	// ===== bw200-C2 =====
	REGION J2.1.2
	    //J2.1.2
	    DB_UDI.EmptyLine.Fault.Stop.Conveyor[_."J2.1.2"] :=
	    _."ASiGW-MCC001-bw200-C2: Input"."Error J2.1.2" OR
	    _."ASiGW-MCC001-bw200-C2: ConfigErr".Slave."16A" OR
	    _."ASiGW-MCC001-bw200-C2: PeriErr".Slave."16A" OR
	    _.Global.IDB_HardwareDiag."BW-ASi -10.106.129.200".CommunicationError;
	    
	END_REGION
	
	// ===== bw200-C2 =====
	REGION J2.1.3
	    //J2.1.3
	    DB_UDI.EmptyLine.Fault.Stop.Conveyor[_."J2.1.3"] :=
	    _."ASiGW-MCC001-bw200-C2: Input"."Error J2.1.3" OR
	    _."ASiGW-MCC001-bw200-C2: ConfigErr".Slave."17A" OR
	    _."ASiGW-MCC001-bw200-C2: PeriErr".Slave."17A" OR
	    _.Global.IDB_HardwareDiag."BW-ASi -10.106.129.200".CommunicationError;
	    
	END_REGION
	
	// ===== bw200-C2 =====
	REGION J2.1.4
	    //J2.1.4
	    DB_UDI.EmptyLine.Fault.Stop.Conveyor[_."J2.1.4"] :=
	    _."ASiGW-MCC001-bw200-C2: Input"."Error J2.1.4" OR
	    _."ASiGW-MCC001-bw200-C2: ConfigErr".Slave."17A" OR
	    _."ASiGW-MCC001-bw200-C2: PeriErr".Slave."17A" OR
	    _.Global.IDB_HardwareDiag."BW-ASi -10.106.129.200".CommunicationError;
	    
	END_REGION
	
	// ===== bw200-C2 =====
	REGION J2.1.5
	    //J2.1.5
	    DB_UDI.EmptyLine.Fault.Stop.Conveyor[_."J2.1.5"] :=
	    _."ASiGW-MCC001-bw200-C2: Input"."Error J2.1.5" OR
	    _."ASiGW-MCC001-bw200-C2: ConfigErr".Slave."18A" OR
	    _."ASiGW-MCC001-bw200-C2: PeriErr".Slave."18A" OR
	    _.Global.IDB_HardwareDiag."BW-ASi -10.106.129.200".CommunicationError;
	    
	END_REGION
	
	// ===== bw200-C2 =====
	REGION J2.1.6
	    //J2.1.6
	    DB_UDI.EmptyLine.Fault.Stop.Conveyor[_."J2.1.6"] :=
	    _."ASiGW-MCC001-bw200-C2: Input"."Error J2.1.6" OR
	    _."ASiGW-MCC001-bw200-C2: ConfigErr".Slave."18A" OR
	    _."ASiGW-MCC001-bw200-C2: PeriErr".Slave."18A" OR
	    _.Global.IDB_HardwareDiag."BW-ASi -10.106.129.200".CommunicationError;
	    
	END_REGION
	
	// ===== bw200-C2 =====
	REGION J2.1.7
	    //J2.1.7
	    DB_UDI.EmptyLine.Fault.Stop.Conveyor[_."J2.1.7"] :=
	    _."ASiGW-MCC001-bw200-C2: Input"."Error J2.1.7" OR
	    _."ASiGW-MCC001-bw200-C2: ConfigErr".Slave."19A" OR
	    _."ASiGW-MCC001-bw200-C2: PeriErr".Slave."19A" OR
	    _.Global.IDB_HardwareDiag."BW-ASi -10.106.129.200".CommunicationError;
	    
	END_REGION
	
	// ===== bw200-C2 =====
	REGION J2.1.8
	    //J2.1.8
	    DB_UDI.EmptyLine.Fault.Stop.Conveyor[_."J2.1.8"] :=
	    _."ASiGW-MCC001-bw200-C2: Input"."Error J2.1.8" OR
	    _."ASiGW-MCC001-bw200-C2: ConfigErr".Slave."19A" OR
	    _."ASiGW-MCC001-bw200-C2: PeriErr".Slave."19A" OR
	    _.Global.IDB_HardwareDiag."BW-ASi -10.106.129.200".CommunicationError;
	    
	END_REGION
	
	// ===== bw200-C2 =====
	REGION J2.1.9
	    //J2.1.9
	    DB_UDI.EmptyLine.Fault.Stop.Conveyor[_."J2.1.9"] :=
	    _."ASiGW-MCC001-bw200-C2: Input"."Error J2.1.9" OR
	    _."ASiGW-MCC001-bw200-C2: ConfigErr".Slave."20A" OR
	    _."ASiGW-MCC001-bw200-C2: PeriErr".Slave."20A" OR
	    _.Global.IDB_HardwareDiag."BW-ASi -10.106.129.200".CommunicationError;
	    
	END_REGION
	
	// ===== bw200-C2 =====
	REGION J2.1.10
	    //J2.1.10
	    DB_UDI.EmptyLine.Fault.Stop.Conveyor[_."J2.1.10"] :=
	    _."ASiGW-MCC001-bw200-C2: Input"."Error J2.1.10" OR
	    _."ASiGW-MCC001-bw200-C2: ConfigErr".Slave."20A" OR
	    _."ASiGW-MCC001-bw200-C2: PeriErr".Slave."20A" OR
	    _.Global.IDB_HardwareDiag."BW-ASi -10.106.129.200".CommunicationError;
	    
	END_REGION
	
	// ===== bw200-C2 =====
	REGION J2.1.11
	    //J2.1.11
	    DB_UDI.EmptyLine.Fault.Stop.Conveyor[_."J2.1.11"] :=
	    _."ASiGW-MCC001-bw200-C2: Input"."Error J2.1.11" OR
	    _."ASiGW-MCC001-bw200-C2: ConfigErr".Slave."21A" OR
	    _."ASiGW-MCC001-bw200-C2: PeriErr".Slave."21A" OR
	    _.Global.IDB_HardwareDiag."BW-ASi -10.106.129.200".CommunicationError;
	    
	END_REGION
	
	// ===== bw200-C2 =====
	REGION J2.1.12
	    //J2.1.12
	    DB_UDI.EmptyLine.Fault.Stop.Conveyor[_."J2.1.12"] :=
	    _."ASiGW-MCC001-bw200-C2: Input"."Error J2.1.12" OR
	    _."ASiGW-MCC001-bw200-C2: ConfigErr".Slave."21A" OR
	    _."ASiGW-MCC001-bw200-C2: PeriErr".Slave."21A" OR
	    _.Global.IDB_HardwareDiag."BW-ASi -10.106.129.200".CommunicationError;
	    
	END_REGION
	
	// ===== bw200-C2 =====
	REGION J2.1.13
	    //J2.1.13
	    DB_UDI.EmptyLine.Fault.Stop.Conveyor[_."J2.1.13"] :=
	    _."ASiGW-MCC001-bw200-C2: Input"."Error J2.1.13" OR
	    _."ASiGW-MCC001-bw200-C2: ConfigErr".Slave."22A" OR
	    _."ASiGW-MCC001-bw200-C2: PeriErr".Slave."22A" OR
	    _.Global.IDB_HardwareDiag."BW-ASi -10.106.129.200".CommunicationError;
	    
	END_REGION
	
	// ===== bw200-C2 =====
	REGION J2.1.14
	    //J2.1.14
	    DB_UDI.EmptyLine.Fault.Stop.Conveyor[_."J2.1.14"] :=
	    _."ASiGW-MCC001-bw200-C2: Input"."Error J2.1.14" OR
	    _."ASiGW-MCC001-bw200-C2: ConfigErr".Slave."22A" OR
	    _."ASiGW-MCC001-bw200-C2: PeriErr".Slave."22A" OR
	    _.Global.IDB_HardwareDiag."BW-ASi -10.106.129.200".CommunicationError;
	    
	END_REGION
	
	// ===== bw200-C2 =====
	REGION J2.1.15
	    //J2.1.15
	    DB_UDI.EmptyLine.Fault.Stop.Conveyor[_."J2.1.15"] :=
	    _."ASiGW-MCC001-bw200-C2: Input"."Error J2.1.15" OR
	    _."ASiGW-MCC001-bw200-C2: ConfigErr".Slave."23A" OR
	    _."ASiGW-MCC001-bw200-C2: PeriErr".Slave."23A" OR
	    _.Global.IDB_HardwareDiag."BW-ASi -10.106.129.200".CommunicationError;
	    
	END_REGION
	
	
	// ===== bw200-C2 =====
	REGION J2.2.1
	    //J2.2.1
	    DB_UDI.EmptyLine.Fault.Stop.Conveyor[_."J2.2.1"] :=
	    _."ASiGW-MCC001-bw200-C2: Input"."Error J2.2.1" OR
	    _."ASiGW-MCC001-bw200-C2: ConfigErr".Slave."23A" OR
	    _."ASiGW-MCC001-bw200-C2: PeriErr".Slave."23A" OR
	    _.Global.IDB_HardwareDiag."BW-ASi -10.106.129.200".CommunicationError;
	    
	END_REGION
	
	// ===== bw200-C2 =====
	REGION J2.2.2
	    //J2.2.2
	    DB_UDI.EmptyLine.Fault.Stop.Conveyor[_."J2.2.2"] :=
	    _."ASiGW-MCC001-bw200-C2: Input"."Error J2.2.2" OR
	    _."ASiGW-MCC001-bw200-C2: ConfigErr".Slave."24A" OR
	    _."ASiGW-MCC001-bw200-C2: PeriErr".Slave."24A" OR
	    _.Global.IDB_HardwareDiag."BW-ASi -10.106.129.200".CommunicationError;
	    
	END_REGION
	
	// ===== bw200-C2 =====
	REGION J2.3.1
	    //J2.3.1
	    DB_UDI.EmptyLine.Fault.Stop.Conveyor[_."J2.3.1"] :=
	    _."ASiGW-MCC001-bw200-C2: ConfigErr".Slave."25A" OR
	    _."ASiGW-MCC001-bw200-C2: PeriErr".Slave."25A" OR
	    _.Global.IDB_HardwareDiag."BW-ASi -10.106.129.200".CommunicationError;
	    
	END_REGION
	
	// ===== bw200-C2 =====
	REGION J2.4.1
	    //J2.4.1 Arm for Merger1
	    DB_UDI.EmptyLine.Fault.Stop.Conveyor[_."J2.4.1"] :=
	    _."ASiGW-MCC001-bw200-C2: Input"."Error J2.4.1" OR
	    _."ASiGW-MCC001-bw200-C2: ConfigErr".Slave."26A" OR
	    _."ASiGW-MCC001-bw200-C2: PeriErr".Slave."26A" OR
	    _.Global.IDB_HardwareDiag."BW-ASi -10.106.129.200".CommunicationError;
	    
	END_REGION
	
	
	// ===== bw143-C1 =====
	REGION J1.2.4 Merger1
	    //J1.2.4 Merger 1
	    DB_UDI.EmptyLine.Fault.Stop.Conveyor[_."J1.2.4"] :=
	    _."ASiGW-MCC001-bw143-C1: Input"."Error J1.2.4" OR
	    _."ASiGW-MCC001-bw143-C1: ConfigErr".Slave."27B" OR
	    _."ASiGW-MCC001-bw143-C1: PeriErr".Slave."27B" OR
	    _.Global.IDB_HardwareDiag."BW-ASi -10.106.129.143".CommunicationError;
	    
	END_REGION
	
	// ===== bw143-C1 =====
	REGION J1.2.5
	    //J1.2.5
	    DB_UDI.EmptyLine.Fault.Stop.Conveyor[_."J1.2.5"] :=
	    _."ASiGW-MCC001-bw143-C1: Input"."Error J1.2.5" OR
	    _."ASiGW-MCC001-bw143-C1: ConfigErr".Slave."27B" OR
	    _."ASiGW-MCC001-bw143-C1: PeriErr".Slave."27B" OR
	    _.Global.IDB_HardwareDiag."BW-ASi -10.106.129.143".CommunicationError;
	    
	END_REGION
	
	
	
	
	
	
	
	
	
	// ===== bw143-C1 =====
	REGION J1.3.1
	    //J1.3.1
	    DB_UDI.EmptyLine.Fault.Stop.Conveyor[_."J1.3.1"] :=
	    _."ASiGW-MCC001-bw143-C1: Input"."Error J1.3.1" OR
	    _."ASiGW-MCC001-bw143-C1: ConfigErr".Slave."17B" OR
	    _."ASiGW-MCC001-bw143-C1: PeriErr".Slave."17B" OR
	    _.Global.IDB_HardwareDiag."BW-ASi -10.106.129.143".CommunicationError;
	    
	END_REGION
	
	// ===== bw143-C1 =====
	REGION J1.3.2
	    //J1.3.2
	    DB_UDI.EmptyLine.Fault.Stop.Conveyor[_."J1.3.2"] :=
	    _."ASiGW-MCC001-bw143-C1: Input"."Error J1.3.2" OR
	    _."ASiGW-MCC001-bw143-C1: ConfigErr".Slave."17B" OR
	    _."ASiGW-MCC001-bw143-C1: PeriErr".Slave."17B" OR
	    _.Global.IDB_HardwareDiag."BW-ASi -10.106.129.143".CommunicationError;
	    
	END_REGION
	
	// ===== bw143-C1 =====
	REGION J1.4.1
	    //J1.4.1
	    DB_UDI.EmptyLine.Fault.Stop.Conveyor[_."J1.4.1"] :=
	    _."ASiGW-MCC001-bw143-C1: Input"."Error J1.4.1" OR
	    _."ASiGW-MCC001-bw143-C1: ConfigErr".Slave."13B" OR
	    _."ASiGW-MCC001-bw143-C1: PeriErr".Slave."13B" OR
	    _.Global.IDB_HardwareDiag."BW-ASi -10.106.129.143".CommunicationError;
	    
	END_REGION
	
	// ===== bw143-C1 =====
	REGION J1.4.2
	    //J1.4.2
	    DB_UDI.EmptyLine.Fault.Stop.Conveyor[_."J1.4.2"] :=
	    _."ASiGW-MCC001-bw143-C1: Input"."Error J1.4.2" OR
	    _."ASiGW-MCC001-bw143-C1: ConfigErr".Slave."13B" OR
	    _."ASiGW-MCC001-bw143-C1: PeriErr".Slave."13B" OR
	    _.Global.IDB_HardwareDiag."BW-ASi -10.106.129.143".CommunicationError;
	    
	END_REGION
	
	// ===== bw143-C1 =====
	REGION J1.4.3
	    //J1.4.3
	    DB_UDI.EmptyLine.Fault.Stop.Conveyor[_."J1.4.3"] :=
	    _."ASiGW-MCC001-bw143-C1: Input"."Error J1.4.3" OR
	    _."ASiGW-MCC001-bw143-C1: ConfigErr".Slave."14B" OR
	    _."ASiGW-MCC001-bw143-C1: PeriErr".Slave."14B" OR
	    _.Global.IDB_HardwareDiag."BW-ASi -10.106.129.143".CommunicationError;
	    
	END_REGION
	
	// ===== bw143-C1 =====
	REGION J1.4.4
	    //J1.4.4
	    DB_UDI.EmptyLine.Fault.Stop.Conveyor[_."J1.4.4"] :=
	    _."ASiGW-MCC001-bw143-C1: Input"."Error J1.4.4" OR
	    _."ASiGW-MCC001-bw143-C1: ConfigErr".Slave."14B" OR
	    _."ASiGW-MCC001-bw143-C1: PeriErr".Slave."14B" OR
	    _.Global.IDB_HardwareDiag."BW-ASi -10.106.129.143".CommunicationError;
	    
	END_REGION
	
	// ===== bw143-C1 =====
	REGION J1.4.5
	    //J1.4.5
	    DB_UDI.EmptyLine.Fault.Stop.Conveyor[_."J1.4.5"] :=
	    _."ASiGW-MCC001-bw143-C1: Input"."Error J1.4.5" OR
	    _."ASiGW-MCC001-bw143-C1: ConfigErr".Slave."15B" OR
	    _."ASiGW-MCC001-bw143-C1: PeriErr".Slave."15B" OR
	    _.Global.IDB_HardwareDiag."BW-ASi -10.106.129.143".CommunicationError;
	    
	END_REGION
	
	// ===== bw143-C1 =====
	REGION J1.4.6
	    //J1.4.6
	    DB_UDI.EmptyLine.Fault.Stop.Conveyor[_."J1.4.6"] :=
	    _."ASiGW-MCC001-bw143-C1: Input"."Error J1.4.6" OR
	    _."ASiGW-MCC001-bw143-C1: ConfigErr".Slave."15B" OR
	    _."ASiGW-MCC001-bw143-C1: PeriErr".Slave."15B" OR
	    _.Global.IDB_HardwareDiag."BW-ASi -10.106.129.143".CommunicationError;
	    
	END_REGION
	
	// ===== bw143-C1 =====
	REGION J1.4.7
	    //J1.4.7
	    DB_UDI.EmptyLine.Fault.Stop.Conveyor[_."J1.4.7"] :=
	    _."ASiGW-MCC001-bw143-C1: Input"."Error J1.4.7" OR
	    _."ASiGW-MCC001-bw143-C1: ConfigErr".Slave."16B" OR
	    _."ASiGW-MCC001-bw143-C1: PeriErr".Slave."16B" OR
	    _.Global.IDB_HardwareDiag."BW-ASi -10.106.129.143".CommunicationError;
	    
	END_REGION
	
	// ===== bw143-C1 =====
	REGION J1.5.1
	    //J1.5.1
	    DB_UDI.EmptyLine.Fault.Stop.Conveyor[_."J1.5.1"] :=
	    _."ASiGW-MCC001-bw143-C1: Input"."Error J1.5.1" OR
	    _."ASiGW-MCC001-bw143-C1: ConfigErr".Slave."16B" OR
	    _."ASiGW-MCC001-bw143-C1: PeriErr".Slave."16B" OR
	    _.Global.IDB_HardwareDiag."BW-ASi -10.106.129.143".CommunicationError;
	    
	END_REGION
	
	// ===== bw143-C1 =====
	REGION J1.5.2
	    //J1.5.2
	    DB_UDI.EmptyLine.Fault.Stop.Conveyor[_."J1.5.2"] :=
	    _."ASiGW-MCC001-bw143-C1: Input"."Error J1.5.2" OR
	    _."ASiGW-MCC001-bw143-C1: ConfigErr".Slave."1B" OR
	    _."ASiGW-MCC001-bw143-C1: PeriErr".Slave."1B" OR
	    _.Global.IDB_HardwareDiag."BW-ASi -10.106.129.143".CommunicationError;
	    
	END_REGION
	
	// ===== bw143-C1 =====
	REGION J1.5.3
	    //J1.5.3
	    DB_UDI.EmptyLine.Fault.Stop.Conveyor[_."J1.5.3"] :=
	    _."ASiGW-MCC001-bw143-C1: Input"."Error J1.5.3" OR
	    _."ASiGW-MCC001-bw143-C1: ConfigErr".Slave."2B" OR
	    _."ASiGW-MCC001-bw143-C1: PeriErr".Slave."2B" OR
	    _.Global.IDB_HardwareDiag."BW-ASi -10.106.129.143".CommunicationError;
	    
	END_REGION
	
	// ===== bw143-C1 =====
	REGION J1.5.4
	    //J1.5.4
	    DB_UDI.EmptyLine.Fault.Stop.Conveyor[_."J1.5.4"] :=
	    _."ASiGW-MCC001-bw143-C1: Input"."Error J1.5.4" OR
	    _."ASiGW-MCC001-bw143-C1: ConfigErr".Slave."2B" OR
	    _."ASiGW-MCC001-bw143-C1: PeriErr".Slave."2B" OR
	    _.Global.IDB_HardwareDiag."BW-ASi -10.106.129.143".CommunicationError;
	    
	END_REGION
	
	REGION J1.6.1 Mabs
	    //J1.6.1 Mabs
	    DB_UDI.EmptyLine.Fault.Stop.Conveyor[_."J1.6.1"] :=
	    _."ASiGW-MCC001-bw143-C1: ConfigErr".Slave."29B" OR
	    _."ASiGW-MCC001-bw143-C1: PeriErr".Slave."29B" OR
	    _."ASiGW-MCC001-bw143-C1: ConfigErr".Slave."30B" OR
	    _."ASiGW-MCC001-bw143-C1: PeriErr".Slave."30B" OR
	    _.Global.IDB_HardwareDiag."BW-ASi -10.106.129.143".CommunicationError;
	    
	END_REGION
	
	REGION J1.6.2 Mabs
	    //J1.6.2 Mabs
	    DB_UDI.EmptyLine.Fault.Stop.Conveyor[_."J1.6.2"] :=
	    _."ASiGW-MCC001-bw143-C1: ConfigErr".Slave."29B" OR
	    _."ASiGW-MCC001-bw143-C1: PeriErr".Slave."29B" OR
	    _."ASiGW-MCC001-bw143-C1: ConfigErr".Slave."30B" OR
	    _."ASiGW-MCC001-bw143-C1: PeriErr".Slave."30B" OR
	    _.Global.IDB_HardwareDiag."BW-ASi -10.106.129.143".CommunicationError;
	    
	END_REGION
	
	// ===== bw143-C1 =====
	REGION J1.7.1
	    //J1.7.1 (Go straight )
	    DB_UDI.EmptyLine.Fault.Stop.Conveyor[_."J1.7.1"] :=
	    _."ASiGW-MCC001-bw143-C1: Input"."Error J1.7.1" OR
	    _."ASiGW-MCC001-bw143-C1: ConfigErr".Slave."3B" OR
	    _."ASiGW-MCC001-bw143-C1: PeriErr".Slave."3B" OR
	    _.Global.IDB_HardwareDiag."BW-ASi -10.106.129.143".CommunicationError;
	    
	END_REGION
	
	// ===== bw143-C1 =====
	REGION J1.7.2
	    //J1.7.2
	    DB_UDI.EmptyLine.Fault.Stop.Conveyor[_."J1.7.2"] :=
	    _."ASiGW-MCC001-bw143-C1: Input"."Error J1.7.2" OR
	    _."ASiGW-MCC001-bw143-C1: ConfigErr".Slave."3B" OR
	    _."ASiGW-MCC001-bw143-C1: PeriErr".Slave."3B" OR
	    _.Global.IDB_HardwareDiag."BW-ASi -10.106.129.143".CommunicationError;
	    
	END_REGION
	
	// ===== bw143-C1 =====
	REGION J1.8.1
	    //J1.8.1
	    DB_UDI.EmptyLine.Fault.Stop.Conveyor[_."J1.8.1"] :=
	    _."ASiGW-MCC001-bw143-C1: Input"."Error J1.8.1" OR
	    _."ASiGW-MCC001-bw143-C1: ConfigErr".Slave."4B" OR
	    _."ASiGW-MCC001-bw143-C1: PeriErr".Slave."4B" OR
	    _.Global.IDB_HardwareDiag."BW-ASi -10.106.129.143".CommunicationError;
	    
	END_REGION
	
	// ===== bw143-C1 =====
	REGION J1.8.2
	    //J1.8.2
	    DB_UDI.EmptyLine.Fault.Stop.Conveyor[_."J1.8.2"] :=
	    _."ASiGW-MCC001-bw143-C1: Input"."Error J1.8.2" OR
	    _."ASiGW-MCC001-bw143-C1: ConfigErr".Slave."4B" OR
	    _."ASiGW-MCC001-bw143-C1: PeriErr".Slave."4B" OR
	    _.Global.IDB_HardwareDiag."BW-ASi -10.106.129.143".CommunicationError;
	    
	END_REGION
	
	// ===== bw143-C1 =====
	REGION J1.9.1
	    //J1.9.1
	    DB_UDI.EmptyLine.Fault.Stop.Conveyor[_."J1.9.1"] :=
	    _."ASiGW-MCC001-bw143-C1: ConfigErr".Slave."5B" OR
	    _."ASiGW-MCC001-bw143-C1: PeriErr".Slave."5B" OR
	    _.Global.IDB_HardwareDiag."BW-ASi -10.106.129.143".CommunicationError;
	    
	END_REGION
	
	// ===== bw143-C1 =====
	REGION J1.10.1
	    //J1.10.1
	    DB_UDI.EmptyLine.Fault.Stop.Conveyor[_."J1.10.1"] :=
	    _."ASiGW-MCC001-bw143-C1: ConfigErr".Slave."5B" OR
	    _."ASiGW-MCC001-bw143-C1: PeriErr".Slave."5B" OR
	    _.Global.IDB_HardwareDiag."BW-ASi -10.106.129.143".CommunicationError;
	    
	END_REGION
	
	// ===== bw143-C1 =====
	REGION J1.11.1
	    //J1.11.1
	    DB_UDI.EmptyLine.Fault.Stop.Conveyor[_."J1.11.1"] :=
	    _."ASiGW-MCC001-bw143-C1: Input"."Error J1.11.1" OR
	    _."ASiGW-MCC001-bw143-C1: ConfigErr".Slave."6B" OR
	    _."ASiGW-MCC001-bw143-C1: PeriErr".Slave."6B" OR
	    _.Global.IDB_HardwareDiag."BW-ASi -10.106.129.143".CommunicationError;
	    
	END_REGION
	
	// ===== bw143-C1 =====
	REGION J1.11.2
	    //J1.11.2
	    DB_UDI.EmptyLine.Fault.Stop.Conveyor[_."J1.11.2"] :=
	    _."ASiGW-MCC001-bw143-C1: Input"."Error J1.11.2" OR
	    _."ASiGW-MCC001-bw143-C1: ConfigErr".Slave."6B" OR
	    _."ASiGW-MCC001-bw143-C1: PeriErr".Slave."6B" OR
	    _.Global.IDB_HardwareDiag."BW-ASi -10.106.129.143".CommunicationError;
	    
	END_REGION
	
	// ===== bw143-C1 =====
	REGION J1.11.3
	    //J1.11.3
	    DB_UDI.EmptyLine.Fault.Stop.Conveyor[_."J1.11.3"] :=
	    _."ASiGW-MCC001-bw143-C1: Input"."Error J1.11.3" OR
	    _."ASiGW-MCC001-bw143-C1: ConfigErr".Slave."7B" OR
	    _."ASiGW-MCC001-bw143-C1: PeriErr".Slave."7B" OR
	    _.Global.IDB_HardwareDiag."BW-ASi -10.106.129.143".CommunicationError;
	    
	END_REGION
	
	// ===== bw143-C1 =====
	REGION J1.11.4
	    //J1.11.4
	    DB_UDI.EmptyLine.Fault.Stop.Conveyor[_."J1.11.4"] :=
	    _."ASiGW-MCC001-bw143-C1: Input"."Error J1.11.4" OR
	    _."ASiGW-MCC001-bw143-C1: ConfigErr".Slave."7B" OR
	    _."ASiGW-MCC001-bw143-C1: PeriErr".Slave."7B" OR
	    _.Global.IDB_HardwareDiag."BW-ASi -10.106.129.143".CommunicationError;
	    
	END_REGION
	
	// ===== bw143-C1 =====
	REGION J1.11.5
	    //J1.11.5
	    DB_UDI.EmptyLine.Fault.Stop.Conveyor[_."J1.11.5"] :=
	    _."ASiGW-MCC001-bw143-C1: Input"."Error J1.11.5" OR
	    _."ASiGW-MCC001-bw143-C1: ConfigErr".Slave."8B" OR
	    _."ASiGW-MCC001-bw143-C1: PeriErr".Slave."8B" OR
	    _.Global.IDB_HardwareDiag."BW-ASi -10.106.129.143".CommunicationError;
	    
	END_REGION
	
	// ===== bw143-C1 =====
	REGION J1.11.6
	    //J1.11.6
	    DB_UDI.EmptyLine.Fault.Stop.Conveyor[_."J1.11.6"] :=
	    _."ASiGW-MCC001-bw143-C1: Input"."Error J1.11.6" OR
	    _."ASiGW-MCC001-bw143-C1: ConfigErr".Slave."8B" OR
	    _."ASiGW-MCC001-bw143-C1: PeriErr".Slave."8B" OR
	    _.Global.IDB_HardwareDiag."BW-ASi -10.106.129.143".CommunicationError;
	    
	END_REGION
	
	// ===== bw143-C1 =====
	REGION J1.11.7
	    //J1.11.7
	    DB_UDI.EmptyLine.Fault.Stop.Conveyor[_."J1.11.7"] :=
	    _."ASiGW-MCC001-bw143-C1: Input"."Error J1.11.7" OR
	    _."ASiGW-MCC001-bw143-C1: ConfigErr".Slave."9B" OR
	    _."ASiGW-MCC001-bw143-C1: PeriErr".Slave."9B" OR
	    _.Global.IDB_HardwareDiag."BW-ASi -10.106.129.143".CommunicationError;
	    
	END_REGION
	
	// ===== bw143-C1 =====
	REGION J1.11.8
	    //J1.11.8
	    DB_UDI.EmptyLine.Fault.Stop.Conveyor[_."J1.11.8"] :=
	    _."ASiGW-MCC001-bw143-C1: Input"."Error J1.11.8" OR
	    _."ASiGW-MCC001-bw143-C1: ConfigErr".Slave."9B" OR
	    _."ASiGW-MCC001-bw143-C1: PeriErr".Slave."9B" OR
	    _.Global.IDB_HardwareDiag."BW-ASi -10.106.129.143".CommunicationError;
	    
	END_REGION
	
	// ===== bw143-C1 =====
	REGION J1.11.9
	    //J1.11.9
	    DB_UDI.EmptyLine.Fault.Stop.Conveyor[_."J1.11.9"] :=
	    _."ASiGW-MCC001-bw143-C1: Input"."Error J1.11.9" OR
	    _."ASiGW-MCC001-bw143-C1: ConfigErr".Slave."10B" OR
	    _."ASiGW-MCC001-bw143-C1: PeriErr".Slave."10B" OR
	    _.Global.IDB_HardwareDiag."BW-ASi -10.106.129.143".CommunicationError;
	    
	END_REGION
	
	// ===== bw143-C1 =====
	REGION J1.11.10
	    //J1.11.10
	    DB_UDI.EmptyLine.Fault.Stop.Conveyor[_."J1.11.10"] :=
	    _."ASiGW-MCC001-bw143-C1: Input"."Error J1.11.10" OR
	    _."ASiGW-MCC001-bw143-C1: ConfigErr".Slave."10B" OR
	    _."ASiGW-MCC001-bw143-C1: PeriErr".Slave."10B" OR
	    _.Global.IDB_HardwareDiag."BW-ASi -10.106.129.143".CommunicationError;
	    
	END_REGION
	
	// ===== bw143-C1 =====
	REGION J1.11.11
	    //J1.11.11
	    DB_UDI.EmptyLine.Fault.Stop.Conveyor[_."J1.11.11"] :=
	    _."ASiGW-MCC001-bw143-C1: Input"."Error J1.11.11" OR
	    _."ASiGW-MCC001-bw143-C1: ConfigErr".Slave."11B" OR
	    _."ASiGW-MCC001-bw143-C1: PeriErr".Slave."11B" OR
	    _.Global.IDB_HardwareDiag."BW-ASi -10.106.129.143".CommunicationError;
	    
	END_REGION
	
	// ===== bw143-C1 =====
	REGION J1.11.12
	    //J1.11.12
	    DB_UDI.EmptyLine.Fault.Stop.Conveyor[_."J1.11.12"] :=
	    _."ASiGW-MCC001-bw143-C1: Input"."Error J1.11.12" OR
	    _."ASiGW-MCC001-bw143-C1: ConfigErr".Slave."11B" OR
	    _."ASiGW-MCC001-bw143-C1: PeriErr".Slave."11B" OR
	    _.Global.IDB_HardwareDiag."BW-ASi -10.106.129.143".CommunicationError;
	    
	END_REGION
	
	// ===== bw143-C1 =====
	REGION J1.11.13
	    //J1.11.13
	    DB_UDI.EmptyLine.Fault.Stop.Conveyor[_."J1.11.13"] :=
	    _."ASiGW-MCC001-bw143-C1: Input"."Error J1.11.13" OR
	    _."ASiGW-MCC001-bw143-C1: ConfigErr".Slave."12B" OR
	    _."ASiGW-MCC001-bw143-C1: PeriErr".Slave."12B" OR
	    _.Global.IDB_HardwareDiag."BW-ASi -10.106.129.143".CommunicationError;
	    
	END_REGION
	
	// ===== bw143-C2 =====
	REGION K1.1.1
	    //K1.1.1  (Go Left)
	    DB_UDI.EmptyLine.Fault.Stop.Conveyor[_."K1.1.1"] :=
	    _."ASiGW-MCC001-bw143-C2: Input"."Error K1.1.1" OR
	    _."ASiGW-MCC001-bw143-C2: ConfigErr".Slave."1B" OR
	    _."ASiGW-MCC001-bw143-C2: PeriErr".Slave."1B" OR
	    _.Global.IDB_HardwareDiag."BW-ASi -10.106.129.143".CommunicationError;
	    
	END_REGION
	
	// ===== bw143-C2 =====
	REGION K1.2.1
	    //K1.2.1
	    DB_UDI.EmptyLine.Fault.Stop.Conveyor[_."K1.2.1"] :=
	    _."ASiGW-MCC001-bw143-C2: ConfigErr".Slave."31A" OR
	    _."ASiGW-MCC001-bw143-C2: PeriErr".Slave."31A" OR
	    _.Global.IDB_HardwareDiag."BW-ASi -10.106.129.143".CommunicationError;
	    
	END_REGION
	
	// ===== bw143-C2 =====
	REGION K1.3.1
	    //K1.3.1
	    DB_UDI.EmptyLine.Fault.Stop.Conveyor[_."K1.3.1"] :=
	    _."ASiGW-MCC001-bw143-C2: Input"."Error K1.3.1" OR
	    _."ASiGW-MCC001-bw143-C2: ConfigErr".Slave."1B" OR
	    _."ASiGW-MCC001-bw143-C2: PeriErr".Slave."1B" OR
	    _.Global.IDB_HardwareDiag."BW-ASi -10.106.129.143".CommunicationError;
	    
	END_REGION
	
	// ===== bw143-C2 =====
	REGION K1.4.1
	    //K1.4.1
	    DB_UDI.EmptyLine.Fault.Stop.Conveyor[_."K1.4.1"] :=
	    _."ASiGW-MCC001-bw143-C2: Input"."Error K1.4.1" OR
	    _."ASiGW-MCC001-bw143-C2: ConfigErr".Slave."2B" OR
	    _."ASiGW-MCC001-bw143-C2: PeriErr".Slave."2B" OR
	    _.Global.IDB_HardwareDiag."BW-ASi -10.106.129.143".CommunicationError;
	    
	END_REGION
	
	// ===== bw143-C2 =====
	REGION K1.4.2
	    //K1.4.2
	    DB_UDI.EmptyLine.Fault.Stop.Conveyor[_."K1.4.2"] :=
	    _."ASiGW-MCC001-bw143-C2: Input"."Error K1.4.2" OR
	    _."ASiGW-MCC001-bw143-C2: ConfigErr".Slave."2B" OR
	    _."ASiGW-MCC001-bw143-C2: PeriErr".Slave."2B" OR
	    _.Global.IDB_HardwareDiag."BW-ASi -10.106.129.143".CommunicationError;
	    
	END_REGION
	
	// ===== bw143-C2 =====
	REGION K1.4.3
	    //K1.4.3
	    DB_UDI.EmptyLine.Fault.Stop.Conveyor[_."K1.4.3"] :=
	    _."ASiGW-MCC001-bw143-C2: Input"."Error K1.4.3" OR
	    _."ASiGW-MCC001-bw143-C2: ConfigErr".Slave."3B" OR
	    _."ASiGW-MCC001-bw143-C2: PeriErr".Slave."3B" OR
	    _.Global.IDB_HardwareDiag."BW-ASi -10.106.129.143".CommunicationError;
	    
	END_REGION
	
	// ===== bw143-C2 =====
	REGION K1.4.4
	    //K1.4.4
	    DB_UDI.EmptyLine.Fault.Stop.Conveyor[_."K1.4.4"] :=
	    _."ASiGW-MCC001-bw143-C2: Input"."Error K1.4.4" OR
	    _."ASiGW-MCC001-bw143-C2: ConfigErr".Slave."3B" OR
	    _."ASiGW-MCC001-bw143-C2: PeriErr".Slave."3B" OR
	    _.Global.IDB_HardwareDiag."BW-ASi -10.106.129.143".CommunicationError;
	    
	END_REGION
	
	// ===== bw143-C2 =====
	REGION K1.4.5
	    //K1.4.5
	    DB_UDI.EmptyLine.Fault.Stop.Conveyor[_."K1.4.5"] :=
	    _."ASiGW-MCC001-bw143-C2: Input"."Error K1.4.5" OR
	    _."ASiGW-MCC001-bw143-C2: ConfigErr".Slave."4B" OR
	    _."ASiGW-MCC001-bw143-C2: PeriErr".Slave."4B" OR
	    _.Global.IDB_HardwareDiag."BW-ASi -10.106.129.143".CommunicationError;
	    
	END_REGION
	
	// ===== bw143-C2 =====
	REGION K1.4.6
	    //K1.4.6
	    DB_UDI.EmptyLine.Fault.Stop.Conveyor[_."K1.4.6"] :=
	    _."ASiGW-MCC001-bw143-C2: Input"."Error K1.4.6" OR
	    _."ASiGW-MCC001-bw143-C2: ConfigErr".Slave."4B" OR
	    _."ASiGW-MCC001-bw143-C2: PeriErr".Slave."4B" OR
	    _.Global.IDB_HardwareDiag."BW-ASi -10.106.129.143".CommunicationError;
	    
	END_REGION
	
	// ===== bw143-C2 =====
	REGION K1.4.7
	    //K1.4.7
	    DB_UDI.EmptyLine.Fault.Stop.Conveyor[_."K1.4.7"] :=
	    _."ASiGW-MCC001-bw143-C2: Input"."Error K1.4.7" OR
	    _."ASiGW-MCC001-bw143-C2: ConfigErr".Slave."5B" OR
	    _."ASiGW-MCC001-bw143-C2: PeriErr".Slave."5B" OR
	    _.Global.IDB_HardwareDiag."BW-ASi -10.106.129.143".CommunicationError;
	    
	END_REGION
	
	// ===== bw143-C2 =====
	REGION K1.4.8
	    //K1.4.8
	    DB_UDI.EmptyLine.Fault.Stop.Conveyor[_."K1.4.8"] :=
	    _."ASiGW-MCC001-bw143-C2: Input"."Error K1.4.8" OR
	    _."ASiGW-MCC001-bw143-C2: ConfigErr".Slave."5B" OR
	    _."ASiGW-MCC001-bw143-C2: PeriErr".Slave."5B" OR
	    _.Global.IDB_HardwareDiag."BW-ASi -10.106.129.143".CommunicationError;
	    
	END_REGION
	
	// ===== bw143-C2 =====
	REGION K1.4.9
	    //K1.4.9
	    DB_UDI.EmptyLine.Fault.Stop.Conveyor[_."K1.4.9"] :=
	    _."ASiGW-MCC001-bw143-C2: Input"."Error K1.4.9" OR
	    _."ASiGW-MCC001-bw143-C2: ConfigErr".Slave."6B" OR
	    _."ASiGW-MCC001-bw143-C2: PeriErr".Slave."6B" OR
	    _.Global.IDB_HardwareDiag."BW-ASi -10.106.129.143".CommunicationError;
	    
	END_REGION
	
	// ===== bw143-C2 =====
	REGION K1.4.10
	    //K1.4.10
	    DB_UDI.EmptyLine.Fault.Stop.Conveyor[_."K1.4.10"] :=
	    _."ASiGW-MCC001-bw143-C2: Input"."Error K1.4.10" OR
	    _."ASiGW-MCC001-bw143-C2: ConfigErr".Slave."6B" OR
	    _."ASiGW-MCC001-bw143-C2: PeriErr".Slave."6B" OR
	    _.Global.IDB_HardwareDiag."BW-ASi -10.106.129.143".CommunicationError;
	    
	END_REGION
	
	// ===== bw143-C2 =====
	REGION K1.5.1
	    //K1.5.1
	    DB_UDI.EmptyLine.Fault.Stop.Conveyor[_."K1.5.1"] :=
	    _."ASiGW-MCC001-bw143-C2: Input"."Error K1.5.1" OR
	    _."ASiGW-MCC001-bw143-C2: ConfigErr".Slave."7B" OR
	    _."ASiGW-MCC001-bw143-C2: PeriErr".Slave."7B" OR
	    _.Global.IDB_HardwareDiag."BW-ASi -10.106.129.143".CommunicationError;
	    
	END_REGION
	
	// ===== bw143-C2 =====
	REGION K1.5.2
	    //K1.5.2
	    DB_UDI.EmptyLine.Fault.Stop.Conveyor[_."K1.5.2"] :=
	    _."ASiGW-MCC001-bw143-C2: Input"."Error K1.5.2" OR
	    _."ASiGW-MCC001-bw143-C2: ConfigErr".Slave."7B" OR
	    _."ASiGW-MCC001-bw143-C2: PeriErr".Slave."7B" OR
	    _.Global.IDB_HardwareDiag."BW-ASi -10.106.129.143".CommunicationError;
	    
	END_REGION
	
	// ===== bw143-C2 =====
	REGION K1.5.3
	    //K1.5.3
	    DB_UDI.EmptyLine.Fault.Stop.Conveyor[_."K1.5.3"] :=
	    _."ASiGW-MCC001-bw143-C2: Input"."Error K1.5.3" OR
	    _."ASiGW-MCC001-bw143-C2: ConfigErr".Slave."8B" OR
	    _."ASiGW-MCC001-bw143-C2: PeriErr".Slave."8B" OR
	    _.Global.IDB_HardwareDiag."BW-ASi -10.106.129.143".CommunicationError;
	    
	END_REGION
	
	// ===== bw143-C2 =====
	REGION K1.5.4
	    //K1.5.4
	    DB_UDI.EmptyLine.Fault.Stop.Conveyor[_."K1.5.4"] :=
	    _."ASiGW-MCC001-bw143-C2: Input"."Error K1.5.4" OR
	    _."ASiGW-MCC001-bw143-C2: ConfigErr".Slave."8B" OR
	    _."ASiGW-MCC001-bw143-C2: PeriErr".Slave."8B" OR
	    _.Global.IDB_HardwareDiag."BW-ASi -10.106.129.143".CommunicationError;
	    
	END_REGION
	
	// ===== bw143-C2 =====
	REGION K1.5.5
	    //K1.5.5
	    DB_UDI.EmptyLine.Fault.Stop.Conveyor[_."K1.5.5"] :=
	    _."ASiGW-MCC001-bw143-C2: Input"."Error K1.5.5" OR
	    _."ASiGW-MCC001-bw143-C2: ConfigErr".Slave."9B" OR
	    _."ASiGW-MCC001-bw143-C2: PeriErr".Slave."9B" OR
	    _.Global.IDB_HardwareDiag."BW-ASi -10.106.129.143".CommunicationError;
	    
	END_REGION
	
	// ===== bw143-C2 =====
	REGION K1.5.6
	    //K1.5.6
	    DB_UDI.EmptyLine.Fault.Stop.Conveyor[_."K1.5.6"] :=
	    _."ASiGW-MCC001-bw143-C2: Input"."Error K1.5.6" OR
	    _."ASiGW-MCC001-bw143-C2: ConfigErr".Slave."9B" OR
	    _."ASiGW-MCC001-bw143-C2: PeriErr".Slave."9B" OR
	    _.Global.IDB_HardwareDiag."BW-ASi -10.106.129.143".CommunicationError;
	    
	END_REGION
	
	// ===== bw143-C2 =====
	REGION K1.5.7
	    //K1.5.7
	    DB_UDI.EmptyLine.Fault.Stop.Conveyor[_."K1.5.7"] :=
	    _."ASiGW-MCC001-bw143-C2: Input"."Error K1.5.7" OR
	    _."ASiGW-MCC001-bw143-C2: ConfigErr".Slave."10B" OR
	    _."ASiGW-MCC001-bw143-C2: PeriErr".Slave."10B" OR
	    _.Global.IDB_HardwareDiag."BW-ASi -10.106.129.143".CommunicationError;
	    
	END_REGION
	
	// ===== bw143-C2 =====
	REGION K1.5.8
	    //K1.5.8
	    DB_UDI.EmptyLine.Fault.Stop.Conveyor[_."K1.5.8"] :=
	    _."ASiGW-MCC001-bw143-C2: Input"."Error K1.5.8" OR
	    _."ASiGW-MCC001-bw143-C2: ConfigErr".Slave."10B" OR
	    _."ASiGW-MCC001-bw143-C2: PeriErr".Slave."10B" OR
	    _.Global.IDB_HardwareDiag."BW-ASi -10.106.129.143".CommunicationError;
	    
	END_REGION
	
	// ===== bw143-C2 =====
	REGION K1.6.1
	    //K1.6.1
	    DB_UDI.EmptyLine.Fault.Stop.Conveyor[_."K1.6.1"] :=
	    _."ASiGW-MCC001-bw143-C2: ConfigErr".Slave."11B" OR
	    _."ASiGW-MCC001-bw143-C2: PeriErr".Slave."11B" OR
	    _.Global.IDB_HardwareDiag."BW-ASi -10.106.129.143".CommunicationError;
	    
	END_REGION
	
	// ===== bw143-C2 =====
	REGION K1.6.2
	    //K1.6.2
	    DB_UDI.EmptyLine.Fault.Stop.Conveyor[_."K1.6.2"] :=
	    _."ASiGW-MCC001-bw143-C2: ConfigErr".Slave."11B" OR
	    _."ASiGW-MCC001-bw143-C2: PeriErr".Slave."11B" OR
	    _.Global.IDB_HardwareDiag."BW-ASi -10.106.129.143".CommunicationError;
	    
	END_REGION
	
	// ===== bw143-C2 =====
	REGION K1.7.1
	    //K1.7.1
	    DB_UDI.EmptyLine.Fault.Stop.Conveyor[_."K1.7.1"] :=
	    _."ASiGW-MCC001-bw143-C2: Input"."Error K1.7.1" OR
	    _."ASiGW-MCC001-bw143-C2: ConfigErr".Slave."12B" OR
	    _."ASiGW-MCC001-bw143-C2: PeriErr".Slave."12B" OR
	    _.Global.IDB_HardwareDiag."BW-ASi -10.106.129.143".CommunicationError;
	    
	END_REGION
	
	// ===== bw143-C2 =====
	REGION K1.7.2
	    //K1.7.2
	    DB_UDI.EmptyLine.Fault.Stop.Conveyor[_."K1.7.2"] :=
	    _."ASiGW-MCC001-bw143-C2: Input"."Error K1.7.2" OR
	    _."ASiGW-MCC001-bw143-C2: ConfigErr".Slave."12B" OR
	    _."ASiGW-MCC001-bw143-C2: PeriErr".Slave."12B" OR
	    _.Global.IDB_HardwareDiag."BW-ASi -10.106.129.143".CommunicationError;
	    
	END_REGION
	
	// ===== bw143-C2 =====
	REGION K1.8.1
	    //K1.8.1
	    DB_UDI.EmptyLine.Fault.Stop.Conveyor[_."K1.8.1"] :=
	    _."ASiGW-MCC001-bw143-C2: Input"."Error K1.8.1" OR
	    _."ASiGW-MCC001-bw143-C2: ConfigErr".Slave."13B" OR
	    _."ASiGW-MCC001-bw143-C2: PeriErr".Slave."13B" OR
	    _.Global.IDB_HardwareDiag."BW-ASi -10.106.129.143".CommunicationError;
	    
	END_REGION
	
	// ===== bw143-C2 =====
	REGION K1.8.2
	    //K1.8.2
	    DB_UDI.EmptyLine.Fault.Stop.Conveyor[_."K1.8.2"] :=
	    _."ASiGW-MCC001-bw143-C2: Input"."Error K1.8.2" OR
	    _."ASiGW-MCC001-bw143-C2: ConfigErr".Slave."13B" OR
	    _."ASiGW-MCC001-bw143-C2: PeriErr".Slave."13B" OR
	    _.Global.IDB_HardwareDiag."BW-ASi -10.106.129.143".CommunicationError;
	    
	END_REGION
	
	// ===== bw143-C2 =====
	REGION K1.8.3
	    //K1.8.3
	    DB_UDI.EmptyLine.Fault.Stop.Conveyor[_."K1.8.3"] :=
	    _."ASiGW-MCC001-bw143-C2: Input"."Error K1.8.3" OR
	    _."ASiGW-MCC001-bw143-C2: ConfigErr".Slave."14B" OR
	    _."ASiGW-MCC001-bw143-C2: PeriErr".Slave."14B" OR
	    _.Global.IDB_HardwareDiag."BW-ASi -10.106.129.143".CommunicationError;
	    
	END_REGION
	
	// ===== bw143-C2 =====
	REGION K1.9.1
	    //K1.9.1
	    DB_UDI.EmptyLine.Fault.Stop.Conveyor[_."K1.9.1"] :=
	    _."ASiGW-MCC001-bw143-C2: Input"."Error K1.9.1" OR
	    _."ASiGW-MCC001-bw143-C2: ConfigErr".Slave."15B" OR
	    _."ASiGW-MCC001-bw143-C2: PeriErr".Slave."15B" OR
	    _.Global.IDB_HardwareDiag."BW-ASi -10.106.129.143".CommunicationError;
	    
	END_REGION
	
	// ===== bw143-C2 =====
	REGION K1.9.2
	    //K1.9.2
	    DB_UDI.EmptyLine.Fault.Stop.Conveyor[_."K1.9.2"] :=
	    _."ASiGW-MCC001-bw143-C2: Input"."Error K1.9.2" OR
	    _."ASiGW-MCC001-bw143-C2: ConfigErr".Slave."15B" OR
	    _."ASiGW-MCC001-bw143-C2: PeriErr".Slave."15B" OR
	    _.Global.IDB_HardwareDiag."BW-ASi -10.106.129.143".CommunicationError;
	    
	END_REGION
	
	// ===== bw143-C2 =====
	REGION K1.9.3
	    //K1.9.3
	    DB_UDI.EmptyLine.Fault.Stop.Conveyor[_."K1.9.3"] :=
	    _."ASiGW-MCC001-bw143-C2: Input"."Error K1.9.3" OR
	    _."ASiGW-MCC001-bw143-C2: ConfigErr".Slave."16B" OR
	    _."ASiGW-MCC001-bw143-C2: PeriErr".Slave."16B" OR
	    _.Global.IDB_HardwareDiag."BW-ASi -10.106.129.143".CommunicationError;
	    
	END_REGION
	
	// ===== bw143-C2 =====
	REGION K1.9.4
	    //K1.9.4
	    DB_UDI.EmptyLine.Fault.Stop.Conveyor[_."K1.9.4"] :=
	    _."ASiGW-MCC001-bw143-C2: Input"."Error K1.9.4" OR
	    _."ASiGW-MCC001-bw143-C2: ConfigErr".Slave."16B" OR
	    _."ASiGW-MCC001-bw143-C2: PeriErr".Slave."16B" OR
	    _.Global.IDB_HardwareDiag."BW-ASi -10.106.129.143".CommunicationError;
	    
	END_REGION
	
	// ===== bw143-C2 =====
	REGION K1.9.5
	    //K1.9.5
	    DB_UDI.EmptyLine.Fault.Stop.Conveyor[_."K1.9.5"] :=
	    _."ASiGW-MCC001-bw143-C2: Input"."Error K1.9.5" OR
	    _."ASiGW-MCC001-bw143-C2: ConfigErr".Slave."17B" OR
	    _."ASiGW-MCC001-bw143-C2: PeriErr".Slave."17B" OR
	    _.Global.IDB_HardwareDiag."BW-ASi -10.106.129.143".CommunicationError;
	    
	END_REGION
	
	// ===== bw143-C2 =====
	REGION K1.9.6
	    //K1.9.6
	    DB_UDI.EmptyLine.Fault.Stop.Conveyor[_."K1.9.6"] :=
	    _."ASiGW-MCC001-bw143-C2: Input"."Error K1.9.6" OR
	    _."ASiGW-MCC001-bw143-C2: ConfigErr".Slave."17B" OR
	    _."ASiGW-MCC001-bw143-C2: PeriErr".Slave."17B" OR
	    _.Global.IDB_HardwareDiag."BW-ASi -10.106.129.143".CommunicationError;
	    
	END_REGION
	
	// ===== bw143-C2 =====
	REGION K1.9.7
	    //K1.9.7
	    DB_UDI.EmptyLine.Fault.Stop.Conveyor[_."K1.9.7"] :=
	    _."ASiGW-MCC001-bw143-C2: Input"."Error K1.9.7" OR
	    _."ASiGW-MCC001-bw143-C2: ConfigErr".Slave."18B" OR
	    _."ASiGW-MCC001-bw143-C2: PeriErr".Slave."18B" OR
	    _.Global.IDB_HardwareDiag."BW-ASi -10.106.129.143".CommunicationError;
	    
	END_REGION
	
	// ===== bw143-C2 =====
	REGION K1.10.1
	    //K1.10.1
	    DB_UDI.EmptyLine.Fault.Stop.Conveyor[_."K1.10.1"] :=
	    _."ASiGW-MCC001-bw143-C2: Input"."Error K1.10.1" OR
	    _."ASiGW-MCC001-bw143-C2: ConfigErr".Slave."19B" OR
	    _."ASiGW-MCC001-bw143-C2: PeriErr".Slave."19B" OR
	    _.Global.IDB_HardwareDiag."BW-ASi -10.106.129.143".CommunicationError;
	    
	END_REGION
	
	
END_FUNCTION
END_NAMESPACE

NAMESPACE EmptyLine
FUNCTION FC_Upstream : Void
{ S7_Optimized_Access := 'TRUE' ; Published := 'TRUE' }
VERSION : 0.1

BEGIN
	// ==========================================================================================================================================
	// Company        : LogTech, s.r.o.
	// Created by     : Anton Vinoth Soundraraj
	// Block          : FC_Upstream
	// Project        : Lékarna DC Chrudim
	// Project number : 23-157
	// ==========================================================================================================================================
	
	REGION J1.1.1
	    //J1.1.1
	    DB_UDI.EmptyLine.Upstream.Conveyor[_."J1.1.1"] :=
	    IDB_EmptyLine."J1.1.1".FilteredSensor;
	    
	END_REGION
	
	REGION J1.1.2
	    //J1.1.2
	    DB_UDI.EmptyLine.Upstream.Conveyor[_."J1.1.2"] :=
	    IDB_EmptyLine."J1.1.1".FilteredSensor;
	    
	END_REGION
	
	REGION J1.1.3 TO J1.1.11
	    REGION J1.1.3
	        //J1.1.3
	        DB_UDI.EmptyLine.Upstream.Conveyor[_."J1.1.3"] :=
	        DB_UDI.EmptyLine.Upstream.Conveyor[_."J1.1.4"];
	        
	    END_REGION
	    
	    REGION J1.1.4
	        //J1.1.4
	        DB_UDI.EmptyLine.Upstream.Conveyor[_."J1.1.4"] :=
	        DB_UDI.EmptyLine.Upstream.Conveyor[_."J1.1.5"];
	        
	    END_REGION
	    
	    REGION J1.1.5
	        //J1.1.5
	        DB_UDI.EmptyLine.Upstream.Conveyor[_."J1.1.5"] :=
	        DB_UDI.EmptyLine.Upstream.Conveyor[_."J1.1.6"];
	        
	    END_REGION
	    
	    REGION J1.1.6
	        //J1.1.6
	        DB_UDI.EmptyLine.Upstream.Conveyor[_."J1.1.6"] :=
	        DB_UDI.EmptyLine.Upstream.Conveyor[_."J1.1.7"];
	        
	    END_REGION
	    
	    REGION J1.1.7
	        //J1.1.7
	        DB_UDI.EmptyLine.Upstream.Conveyor[_."J1.1.7"] :=
	        DB_UDI.EmptyLine.Upstream.Conveyor[_."J1.1.8"];
	        
	    END_REGION
	    
	    REGION J1.1.8
	        //J1.1.8
	        DB_UDI.EmptyLine.Upstream.Conveyor[_."J1.1.8"] :=
	        DB_UDI.EmptyLine.Upstream.Conveyor[_."J1.1.9"];
	        
	    END_REGION
	    
	    REGION J1.1.9
	        //J1.1.9
	        DB_UDI.EmptyLine.Upstream.Conveyor[_."J1.1.9"] :=
	        DB_UDI.EmptyLine.Upstream.Conveyor[_."J1.1.10"];
	        
	    END_REGION
	    
	    REGION J1.1.10
	        //J1.1.10
	        DB_UDI.EmptyLine.Upstream.Conveyor[_."J1.1.10"] :=
	        DB_UDI.EmptyLine.Upstream.Conveyor[_."J1.1.11"];
	        
	    END_REGION
	    
	    REGION J1.1.11
	        //J1.1.11
	        DB_UDI.EmptyLine.Upstream.Conveyor[_."J1.1.11"] :=
	        IDB_EmptyLine."J1.1.2".FilteredSensor OR
	        _."ASiGW-MCC001-bw143-C1: Input"."Sensor J1.1.3/J1.1.7-BG1(R-T)-R" OR
	        _."ASiGW-MCC001-bw143-C1: Input"."Sensor J1.1.7/J1.1.11-BG1(R-T)-R";
	        
	    END_REGION
	END_REGION
	
	
	REGION J1.1.12 TO J1.1.15 
	    REGION J1.1.12
	        //J1.1.12
	        DB_UDI.EmptyLine.Upstream.Conveyor[_."J1.1.12"] :=
	        DB_UDI.EmptyLine.Upstream.Conveyor[_."J1.1.13"];
	        
	    END_REGION
	    
	    REGION J1.1.13
	        //J1.1.13
	        DB_UDI.EmptyLine.Upstream.Conveyor[_."J1.1.13"] :=
	        DB_UDI.EmptyLine.Upstream.Conveyor[_."J1.1.14"];
	        
	    END_REGION
	    
	    REGION J1.1.14
	        //J1.1.14
	        DB_UDI.EmptyLine.Upstream.Conveyor[_."J1.1.14"] :=
	        DB_UDI.EmptyLine.Upstream.Conveyor[_."J1.1.15"];
	        
	    END_REGION
	    
	    REGION J1.1.15
	        //J1.1.15
	        DB_UDI.EmptyLine.Upstream.Conveyor[_."J1.1.15"] :=
	        IDB_EmptyLine."J1.1.11".FilteredSensor;
	        
	    END_REGION
	END_REGION
	
	
	REGION J1.2.1
	    //J1.2.1
	    DB_UDI.EmptyLine.Upstream.Conveyor[_."J1.2.1"] :=
	    IDB_EmptyLine."J1.1.15".FilteredSensor;
	    
	END_REGION
	
	REGION J1.2.2
	    //J1.2.2
	    DB_UDI.EmptyLine.Upstream.Conveyor[_."J1.2.2"] :=
	    IDB_EmptyLine."J1.2.1".FilteredSensor;
	    
	END_REGION
	
	REGION J1.2.3
	    //J1.2.3 Staright for Merger1
	    DB_UDI.EmptyLine.Upstream.Conveyor[_."J1.2.3"] :=
	    IDB_EmptyLine."J1.2.2".FilteredSensor;
	    
	END_REGION
	
	REGION J2.1.1 Straight
	    //J2.1.1
	    DB_UDI.EmptyLine.Upstream.Conveyor[_."J2.1.1"] :=
	    IDB_EmptyLine."J1.2.3".FilteredSensor;
	    
	END_REGION
	
	REGION J2.1.2
	    //J2.1.2
	    DB_UDI.EmptyLine.Upstream.Conveyor[_."J2.1.2"] :=
	    IDB_EmptyLine."J2.1.1".FilteredSensor;
	    
	END_REGION
	
	REGION J2.1.3 TO J2.1.11
	    REGION J2.1.3
	        //J2.1.3
	        DB_UDI.EmptyLine.Upstream.Conveyor[_."J2.1.3"] :=
	        DB_UDI.EmptyLine.Upstream.Conveyor[_."J2.1.4"];
	        
	    END_REGION
	    
	    REGION J2.1.4
	        //J2.1.4
	        DB_UDI.EmptyLine.Upstream.Conveyor[_."J2.1.4"] :=
	        DB_UDI.EmptyLine.Upstream.Conveyor[_."J2.1.5"];
	        
	    END_REGION
	    
	    REGION J2.1.5
	        //J2.1.5
	        DB_UDI.EmptyLine.Upstream.Conveyor[_."J2.1.5"] :=
	        DB_UDI.EmptyLine.Upstream.Conveyor[_."J2.1.6"];
	        
	    END_REGION
	    
	    REGION J2.1.6
	        //J2.1.6
	        DB_UDI.EmptyLine.Upstream.Conveyor[_."J2.1.6"] :=
	        DB_UDI.EmptyLine.Upstream.Conveyor[_."J2.1.7"];
	        
	    END_REGION
	    
	    REGION J2.1.7
	        //J2.1.7
	        DB_UDI.EmptyLine.Upstream.Conveyor[_."J2.1.7"] :=
	        DB_UDI.EmptyLine.Upstream.Conveyor[_."J2.1.8"];
	        
	    END_REGION
	    
	    REGION J2.1.8
	        //J2.1.8
	        DB_UDI.EmptyLine.Upstream.Conveyor[_."J2.1.8"] :=
	        DB_UDI.EmptyLine.Upstream.Conveyor[_."J2.1.9"];
	        
	    END_REGION
	    
	    REGION J2.1.9
	        //J2.1.9
	        DB_UDI.EmptyLine.Upstream.Conveyor[_."J2.1.9"] :=
	        DB_UDI.EmptyLine.Upstream.Conveyor[_."J2.1.10"];
	        
	    END_REGION
	    
	    REGION J2.1.10
	        //J2.1.10
	        DB_UDI.EmptyLine.Upstream.Conveyor[_."J2.1.10"] :=
	        DB_UDI.EmptyLine.Upstream.Conveyor[_."J2.1.11"];
	        
	    END_REGION
	    
	    REGION J2.1.11
	        //J2.1.11
	        DB_UDI.EmptyLine.Upstream.Conveyor[_."J2.1.11"] :=
	        IDB_EmptyLine."J2.1.2".FilteredSensor OR
	        _."ASiGW-MCC001-bw200-C2: Input"."Sensor J2.1.3/J2.1.7-BG1(R-T)-R" OR
	        _."ASiGW-MCC001-bw200-C2: Input"."Sensor J2.1.7/J2.1.11-BG1(R-T)-R";
	        
	    END_REGION
	END_REGION
	
	
	REGION J2.1.12 TO J2.1.15 
	    REGION J2.1.12
	        //J2.1.12
	        DB_UDI.EmptyLine.Upstream.Conveyor[_."J2.1.12"] :=
	        DB_UDI.EmptyLine.Upstream.Conveyor[_."J2.1.13"];
	        
	    END_REGION
	    
	    REGION J2.1.13
	        //J2.1.13
	        DB_UDI.EmptyLine.Upstream.Conveyor[_."J2.1.13"] :=
	        DB_UDI.EmptyLine.Upstream.Conveyor[_."J2.1.14"];
	        
	    END_REGION
	    
	    REGION J2.1.14
	        //J2.1.14
	        DB_UDI.EmptyLine.Upstream.Conveyor[_."J2.1.14"] :=
	        DB_UDI.EmptyLine.Upstream.Conveyor[_."J2.1.15"];
	        
	    END_REGION
	    
	    REGION J2.1.15
	        //J2.1.15
	        DB_UDI.EmptyLine.Upstream.Conveyor[_."J2.1.15"] :=
	        IDB_EmptyLine."J2.1.11".FilteredSensor OR
	        _."ASiGW-MCC001-bw200-C2: Input"."Sensor J2.1.11/J2.1.15-BG1(R-T)-R";
	        
	    END_REGION
	END_REGION
	
	
	REGION J2.2.1
	    //J2.2.1
	    DB_UDI.EmptyLine.Upstream.Conveyor[_."J2.2.1"] :=
	    IDB_EmptyLine."J2.1.15".FilteredSensor;
	    
	END_REGION
	
	REGION J2.2.2
	    //J2.2.2
	    DB_UDI.EmptyLine.Upstream.Conveyor[_."J2.2.2"] :=
	    IDB_EmptyLine."J2.2.1".FilteredSensor;
	    
	END_REGION
	
	REGION J2.3.1
	    //J2.3.1
	    DB_UDI.EmptyLine.Upstream.Conveyor[_."J2.3.1"] :=
	    IDB_EmptyLine."J2.2.2".FilteredSensor;
	    
	END_REGION
	
	REGION J2.4.1 Arm
	    //J2.4.1 Arm for Merger1
	    DB_UDI.EmptyLine.Upstream.Conveyor[_."J2.4.1"] :=
	    IDB_EmptyLine."J2.3.1".FilteredSensor AND
	    IDB_Merging."Merge_J1.2.4".Priority.Arm;
	    
	END_REGION
	
	REGION J1.2.4 Merger
	    //J1.2.4 Merger 1
	    DB_UDI.EmptyLine.Upstream.Conveyor[_."J1.2.4"] :=
	    IDB_EmptyLine."J2.4.1".FilteredSensor;
	    
	END_REGION
	
	REGION J1.2.5
	    //J1.2.5
	    DB_UDI.EmptyLine.Upstream.Conveyor[_."J1.2.5"] :=
	    IDB_EmptyLine."J1.2.4".FilteredSensor;
	    
	END_REGION
	
	REGION J1.3.1 TO J1.4.7
	    REGION J1.3.1
	        //J1.3.1
	        DB_UDI.EmptyLine.Upstream.Conveyor[_."J1.3.1"] :=
	        DB_UDI.EmptyLine.Upstream.Conveyor[_."J1.3.2"];
	        
	    END_REGION
	    
	    REGION J1.3.2
	        //J1.3.2
	        DB_UDI.EmptyLine.Upstream.Conveyor[_."J1.3.2"] :=
	        DB_UDI.EmptyLine.Upstream.Conveyor[_."J1.4.1"];
	        
	    END_REGION
	    
	    REGION J1.4.1
	        //J1.4.1
	        DB_UDI.EmptyLine.Upstream.Conveyor[_."J1.4.1"] :=
	        DB_UDI.EmptyLine.Upstream.Conveyor[_."J1.4.2"];
	        
	    END_REGION
	    
	    REGION J1.4.2
	        //J1.4.2
	        DB_UDI.EmptyLine.Upstream.Conveyor[_."J1.4.2"] :=
	        DB_UDI.EmptyLine.Upstream.Conveyor[_."J1.4.3"];
	        
	    END_REGION
	    
	    REGION J1.4.3
	        //J1.4.3
	        DB_UDI.EmptyLine.Upstream.Conveyor[_."J1.4.3"] :=
	        DB_UDI.EmptyLine.Upstream.Conveyor[_."J1.4.4"];
	        
	    END_REGION
	    
	    REGION J1.4.4
	        //J1.4.4
	        DB_UDI.EmptyLine.Upstream.Conveyor[_."J1.4.4"] :=
	        DB_UDI.EmptyLine.Upstream.Conveyor[_."J1.4.5"];
	        
	    END_REGION
	    
	    REGION J1.4.5
	        //J1.4.5
	        DB_UDI.EmptyLine.Upstream.Conveyor[_."J1.4.5"] :=
	        DB_UDI.EmptyLine.Upstream.Conveyor[_."J1.4.6"];
	        
	    END_REGION
	    
	    REGION J1.4.6
	        //J1.4.6
	        DB_UDI.EmptyLine.Upstream.Conveyor[_."J1.4.6"] :=
	        DB_UDI.EmptyLine.Upstream.Conveyor[_."J1.4.7"];
	        
	    END_REGION
	    
	    REGION J1.4.7
	        //J1.4.7
	        DB_UDI.EmptyLine.Upstream.Conveyor[_."J1.4.7"] :=
	        IDB_EmptyLine."J1.2.5".FilteredSensor;
	        
	    END_REGION
	END_REGION
	
	
	REGION J1.5.1
	    //J1.5.1
	    DB_UDI.EmptyLine.Upstream.Conveyor[_."J1.5.1"] :=
	    IDB_EmptyLine."J1.4.7".FilteredSensor;
	    
	END_REGION
	
	REGION J1.5.2
	    //J1.5.2
	    DB_UDI.EmptyLine.Upstream.Conveyor[_."J1.5.2"] :=
	    IDB_EmptyLine."J1.5.1".FilteredSensor;
	    
	END_REGION
	
	REGION J1.5.3
	    //J1.5.3
	    DB_UDI.EmptyLine.Upstream.Conveyor[_."J1.5.3"] :=
	    IDB_EmptyLine."J1.5.2".FilteredSensor;
	    
	END_REGION
	
	REGION J1.5.4
	    //J1.5.4
	    DB_UDI.EmptyLine.Upstream.Conveyor[_."J1.5.4"] :=
	    IDB_EmptyLine."J1.5.3".FilteredSensor;
	    
	END_REGION
	
	(* REGION J1.6.1
	    //Mabs J1.6.1
	    DB_UDI.EmptyLine.Upstream.Conveyor[_."J1.6.1"] :=
	    IDB_EmptyLine."J1.5.4".FilteredSensor;
	    
	END_REGION
	
	REGION J1.6.2
	    //Mabs J1.6.2
	    DB_UDI.EmptyLine.Upstream.Conveyor[_."J1.6.2"] :=
	    IDB_EmptyLine."J1.6.1".FilteredSensor;
	    
	END_REGION *)
	
	REGION J1.7.1
	    //J1.7.1 (Go straight )
	    DB_UDI.EmptyLine.Upstream.Conveyor[_."J1.7.1"] :=
	    IDB_EmptyLine."J1.5.4".FilteredSensor AND
	    ToteDir.Conveyor[_."J1.6.1"].Straight AND
	    ToteDir.Conveyor[_."J1.6.2"].Straight;
	    
	END_REGION
	
	REGION J1.7.2
	    //J1.7.2
	    DB_UDI.EmptyLine.Upstream.Conveyor[_."J1.7.2"] :=
	    IDB_EmptyLine."J1.7.1".FilteredSensor;
	    
	END_REGION
	
	REGION J1.8.1
	    //J1.8.1
	    DB_UDI.EmptyLine.Upstream.Conveyor[_."J1.8.1"] :=
	    IDB_EmptyLine."J1.7.2".FilteredSensor;
	    
	END_REGION
	
	REGION J1.8.2
	    //J1.8.2
	    DB_UDI.EmptyLine.Upstream.Conveyor[_."J1.8.2"] :=
	    IDB_EmptyLine."J1.8.1".FilteredSensor;
	    
	END_REGION
	
	REGION J1.9.1
	    //J1.9.1
	    DB_UDI.EmptyLine.Upstream.Conveyor[_."J1.9.1"] :=
	    IDB_EmptyLine."J1.8.2".FilteredSensor;
	    
	END_REGION
	
	REGION J1.10.1
	    //J1.10.1
	    DB_UDI.EmptyLine.Upstream.Conveyor[_."J1.10.1"] :=
	    IDB_EmptyLine."J1.9.1".FilteredSensor;
	    
	END_REGION
	
	REGION J1.11.1 TO J1.11.7
	    REGION J1.11.1
	        //J1.11.1
	        DB_UDI.EmptyLine.Upstream.Conveyor[_."J1.11.1"] :=
	        DB_UDI.EmptyLine.Upstream.Conveyor[_."J1.11.2"];
	        
	    END_REGION
	    
	    REGION J1.11.2
	        //J1.11.2
	        DB_UDI.EmptyLine.Upstream.Conveyor[_."J1.11.2"] :=
	        DB_UDI.EmptyLine.Upstream.Conveyor[_."J1.11.3"];
	        
	    END_REGION
	    
	    REGION J1.11.3
	        //J1.11.3
	        DB_UDI.EmptyLine.Upstream.Conveyor[_."J1.11.3"] :=
	        DB_UDI.EmptyLine.Upstream.Conveyor[_."J1.11.4"];
	        
	    END_REGION
	    
	    REGION J1.11.4
	        //J1.11.4
	        DB_UDI.EmptyLine.Upstream.Conveyor[_."J1.11.4"] :=
	        DB_UDI.EmptyLine.Upstream.Conveyor[_."J1.11.5"];
	        
	    END_REGION
	    
	    REGION J1.11.5
	        //J1.11.5
	        DB_UDI.EmptyLine.Upstream.Conveyor[_."J1.11.5"] :=
	        DB_UDI.EmptyLine.Upstream.Conveyor[_."J1.11.6"];
	        
	    END_REGION
	    
	    REGION J1.11.6
	        //J1.11.6
	        DB_UDI.EmptyLine.Upstream.Conveyor[_."J1.11.6"] :=
	        DB_UDI.EmptyLine.Upstream.Conveyor[_."J1.11.7"];
	        
	    END_REGION
	    
	    REGION J1.11.7
	        //J1.11.7
	        DB_UDI.EmptyLine.Upstream.Conveyor[_."J1.11.7"] :=
	        IDB_EmptyLine."J1.10.1".FilteredSensor;
	        
	    END_REGION
	END_REGION
	
	
	REGION J1.11.8 TO J1.11.13
	    REGION J1.11.8
	        //J1.11.8
	        DB_UDI.EmptyLine.Upstream.Conveyor[_."J1.11.8"] :=
	        DB_UDI.EmptyLine.Upstream.Conveyor[_."J1.11.9"];
	        
	    END_REGION
	    
	    REGION J1.11.9
	        //J1.11.9
	        DB_UDI.EmptyLine.Upstream.Conveyor[_."J1.11.9"] :=
	        DB_UDI.EmptyLine.Upstream.Conveyor[_."J1.11.10"];
	        
	    END_REGION
	    
	    REGION J1.11.10
	        //J1.11.10
	        DB_UDI.EmptyLine.Upstream.Conveyor[_."J1.11.10"] :=
	        DB_UDI.EmptyLine.Upstream.Conveyor[_."J1.11.11"];
	        
	    END_REGION
	    
	    REGION J1.11.11
	        //J1.11.11
	        DB_UDI.EmptyLine.Upstream.Conveyor[_."J1.11.11"] :=
	        DB_UDI.EmptyLine.Upstream.Conveyor[_."J1.11.12"];
	        
	    END_REGION
	    
	    REGION J1.11.12
	        //J1.11.12
	        DB_UDI.EmptyLine.Upstream.Conveyor[_."J1.11.12"] :=
	        DB_UDI.EmptyLine.Upstream.Conveyor[_."J1.11.13"];
	        
	    END_REGION
	    
	    REGION J1.11.13
	        //J1.11.13
	        DB_UDI.EmptyLine.Upstream.Conveyor[_."J1.11.13"] :=
	        IDB_EmptyLine."J1.11.7".FilteredSensor;
	        
	    END_REGION
	END_REGION
	
	
	REGION K1.1.1 TO K1.2.1
	    REGION K1.1.1
	        //K1.1.1  (Go Left)
	        DB_UDI.EmptyLine.Upstream.Conveyor[_."K1.1.1"] :=
	        DB_UDI.EmptyLine.Upstream.Conveyor[_."K1.2.1"];
	        
	    END_REGION
	    
	    REGION K1.2.1
	        //K1.2.1
	        DB_UDI.EmptyLine.Upstream.Conveyor[_."K1.2.1"] :=
	        IDB_EmptyLine."J1.5.4".FilteredSensor AND
	        ToteDir.Conveyor[_."J1.6.1"].toLeft AND
	        ToteDir.Conveyor[_."J1.6.2"].toLeft;
	        
	    END_REGION
	END_REGION
	
	
	REGION K1.3.1
	    //K1.3.1
	    DB_UDI.EmptyLine.Upstream.Conveyor[_."K1.3.1"] :=
	    IDB_EmptyLine."K1.2.1".FilteredSensor;
	    
	END_REGION
	
	REGION K1.4.1
	    //K1.4.1
	    DB_UDI.EmptyLine.Upstream.Conveyor[_."K1.4.1"] :=
	    IDB_EmptyLine."K1.3.1".FilteredSensor;
	    
	END_REGION
	
	REGION K1.4.2 TO K1.4.10
	    REGION K1.4.2
	        //K1.4.2
	        DB_UDI.EmptyLine.Upstream.Conveyor[_."K1.4.2"] :=
	        DB_UDI.EmptyLine.Upstream.Conveyor[_."K1.4.3"];
	        
	    END_REGION
	    
	    REGION K1.4.3
	        //K1.4.3
	        DB_UDI.EmptyLine.Upstream.Conveyor[_."K1.4.3"] :=
	        DB_UDI.EmptyLine.Upstream.Conveyor[_."K1.4.4"];
	        
	    END_REGION
	    
	    REGION K1.4.4
	        //K1.4.4
	        DB_UDI.EmptyLine.Upstream.Conveyor[_."K1.4.4"] :=
	        DB_UDI.EmptyLine.Upstream.Conveyor[_."K1.4.5"];
	        
	    END_REGION
	    
	    REGION K1.4.5
	        //K1.4.5
	        DB_UDI.EmptyLine.Upstream.Conveyor[_."K1.4.5"] :=
	        DB_UDI.EmptyLine.Upstream.Conveyor[_."K1.4.6"];
	        
	    END_REGION
	    
	    REGION K1.4.6
	        //K1.4.6
	        DB_UDI.EmptyLine.Upstream.Conveyor[_."K1.4.6"] :=
	        DB_UDI.EmptyLine.Upstream.Conveyor[_."K1.4.7"];
	        
	    END_REGION
	    
	    REGION K1.4.7
	        //K1.4.7
	        DB_UDI.EmptyLine.Upstream.Conveyor[_."K1.4.7"] :=
	        DB_UDI.EmptyLine.Upstream.Conveyor[_."K1.4.8"];
	        
	    END_REGION
	    
	    REGION K1.4.8
	        //K1.4.8
	        DB_UDI.EmptyLine.Upstream.Conveyor[_."K1.4.8"] :=
	        DB_UDI.EmptyLine.Upstream.Conveyor[_."K1.4.9"];
	        
	    END_REGION
	    
	    REGION K1.4.9
	        //K1.4.9
	        DB_UDI.EmptyLine.Upstream.Conveyor[_."K1.4.9"] :=
	        DB_UDI.EmptyLine.Upstream.Conveyor[_."K1.4.10"];
	        
	    END_REGION
	    
	    REGION K1.4.10
	        //K1.4.10
	        DB_UDI.EmptyLine.Upstream.Conveyor[_."K1.4.10"] :=
	        IDB_EmptyLine."K1.4.1".FilteredSensor;
	        
	    END_REGION
	END_REGION
	
	REGION K1.5.1 TO K1.5.8
	    REGION K1.5.1
	        //K1.5.1
	        DB_UDI.EmptyLine.Upstream.Conveyor[_."K1.5.1"] :=
	        DB_UDI.EmptyLine.Upstream.Conveyor[_."K1.5.2"];
	        
	    END_REGION
	    
	    REGION K1.5.2
	        //K1.5.2
	        DB_UDI.EmptyLine.Upstream.Conveyor[_."K1.5.2"] :=
	        DB_UDI.EmptyLine.Upstream.Conveyor[_."K1.5.3"];
	        
	    END_REGION
	    
	    REGION K1.5.3
	        //K1.5.3
	        DB_UDI.EmptyLine.Upstream.Conveyor[_."K1.5.3"] :=
	        DB_UDI.EmptyLine.Upstream.Conveyor[_."K1.5.4"];
	        
	    END_REGION
	    
	    REGION K1.5.4
	        //K1.5.4
	        DB_UDI.EmptyLine.Upstream.Conveyor[_."K1.5.4"] :=
	        DB_UDI.EmptyLine.Upstream.Conveyor[_."K1.5.5"];
	        
	    END_REGION
	    
	    REGION K1.5.5
	        //K1.5.5
	        DB_UDI.EmptyLine.Upstream.Conveyor[_."K1.5.5"] :=
	        DB_UDI.EmptyLine.Upstream.Conveyor[_."K1.5.6"];
	        
	    END_REGION
	    
	    REGION K1.5.6
	        //K1.5.6
	        DB_UDI.EmptyLine.Upstream.Conveyor[_."K1.5.6"] :=
	        DB_UDI.EmptyLine.Upstream.Conveyor[_."K1.5.7"];
	        
	    END_REGION
	    
	    REGION K1.5.7
	        //K1.5.7
	        DB_UDI.EmptyLine.Upstream.Conveyor[_."K1.5.7"] :=
	        DB_UDI.EmptyLine.Upstream.Conveyor[_."K1.5.8"];
	        
	    END_REGION
	    
	    REGION K1.5.8
	        //K1.5.8
	        DB_UDI.EmptyLine.Upstream.Conveyor[_."K1.5.8"] :=
	        IDB_EmptyLine."K1.4.10".FilteredSensor;
	        
	    END_REGION
	END_REGION
	
	
	REGION K1.6.1
	    //K1.6.1
	    DB_UDI.EmptyLine.Upstream.Conveyor[_."K1.6.1"] :=
	    IDB_EmptyLine."K1.5.8".FilteredSensor;
	    
	END_REGION
	
	REGION K1.6.2
	    //K1.6.2
	    DB_UDI.EmptyLine.Upstream.Conveyor[_."K1.6.2"] :=
	    IDB_EmptyLine."K1.6.1".FilteredSensor;
	    
	END_REGION
	
	REGION K1.7.1 TO K1.7.2
	    REGION K1.7.1
	        //K1.7.1
	        DB_UDI.EmptyLine.Upstream.Conveyor[_."K1.7.1"] :=
	        DB_UDI.EmptyLine.Upstream.Conveyor[_."K1.7.2"];
	        
	    END_REGION
	    
	    REGION K1.7.2
	        //K1.7.2
	        DB_UDI.EmptyLine.Upstream.Conveyor[_."K1.7.2"] :=
	        IDB_EmptyLine."K1.6.2".FilteredSensor;
	        
	    END_REGION
	END_REGION
	
	
	REGION K1.8.1 TO K1.8.3
	    REGION K1.8.1
	        //K1.8.1
	        DB_UDI.EmptyLine.Upstream.Conveyor[_."K1.8.1"] :=
	        DB_UDI.EmptyLine.Upstream.Conveyor[_."K1.8.2"];
	        
	    END_REGION
	    
	    REGION K1.8.2
	        //K1.8.2
	        DB_UDI.EmptyLine.Upstream.Conveyor[_."K1.8.2"] :=
	        DB_UDI.EmptyLine.Upstream.Conveyor[_."K1.8.3"];
	        
	    END_REGION
	    
	    REGION K1.8.3
	        //K1.8.3
	        DB_UDI.EmptyLine.Upstream.Conveyor[_."K1.8.3"] :=
	        IDB_EmptyLine."K1.7.2".FilteredSensor;
	        
	    END_REGION
	END_REGION
	
	
	REGION K1.9.1 TO K1.10.1
	    REGION K1.9.1
	        //K1.9.1
	        DB_UDI.EmptyLine.Upstream.Conveyor[_."K1.9.1"] :=
	        DB_UDI.EmptyLine.Upstream.Conveyor[_."K1.9.2"];
	        
	    END_REGION
	    
	    REGION K1.9.2
	        //K1.9.2
	        DB_UDI.EmptyLine.Upstream.Conveyor[_."K1.9.2"] :=
	        DB_UDI.EmptyLine.Upstream.Conveyor[_."K1.9.3"];
	        
	    END_REGION
	    
	    REGION K1.9.3
	        //K1.9.3
	        DB_UDI.EmptyLine.Upstream.Conveyor[_."K1.9.3"] :=
	        DB_UDI.EmptyLine.Upstream.Conveyor[_."K1.9.4"];
	        
	    END_REGION
	    
	    REGION K1.9.4
	        //K1.9.4
	        DB_UDI.EmptyLine.Upstream.Conveyor[_."K1.9.4"] :=
	        DB_UDI.EmptyLine.Upstream.Conveyor[_."K1.9.5"];
	        
	    END_REGION
	    
	    REGION K1.9.5
	        //K1.9.5
	        DB_UDI.EmptyLine.Upstream.Conveyor[_."K1.9.5"] :=
	        DB_UDI.EmptyLine.Upstream.Conveyor[_."K1.9.6"];
	        
	    END_REGION
	    
	    REGION K1.9.6
	        //K1.9.6
	        DB_UDI.EmptyLine.Upstream.Conveyor[_."K1.9.6"] :=
	        DB_UDI.EmptyLine.Upstream.Conveyor[_."K1.9.7"];
	        
	    END_REGION
	    
	    REGION K1.9.7
	        //K1.9.7
	        DB_UDI.EmptyLine.Upstream.Conveyor[_."K1.9.7"] :=
	        DB_UDI.EmptyLine.Upstream.Conveyor[_."K1.10.1"];
	        
	    END_REGION
	    
	    REGION K1.10.1
	        //K1.10.1
	        DB_UDI.EmptyLine.Upstream.Conveyor[_."K1.10.1"] :=
	        IDB_EmptyLine."K1.8.3".FilteredSensor;
	        
	    END_REGION
	END_REGION
	
	
	
	
END_FUNCTION
END_NAMESPACE

NAMESPACE EmptyLine
FUNCTION FC_Alarm : Void
{ S7_Optimized_Access := 'TRUE' ; Published := 'TRUE' }
VERSION : 0.1

BEGIN
	// ==========================================================================================================================================
	// Company        : LogTech, s.r.o.
	// Created by     : Anton Vinoth Soundraraj
	// Block          : FC_Alarm
	// Project        : Lékarna DC Chrudim
	// Project number : 23-157
	// ==========================================================================================================================================
	
	REGION ASI
	    IF NOT _.Global.IDB_VisuAlarm.noAlarmState THEN
	        
	        // ===== bw143-C1 =====
	        REGION J1.1.1
	            //J1.1.1
	            _.Global.DB_Alarm."word".Line.EmptyLine.Conveyor[_."J1.1.1"].%X1 :=
	            _."ASiGW-MCC001-bw143-C1: Input"."Error J1.1.1";
	            
	        END_REGION
	        
	        // ===== bw143-C1 =====
	        REGION J1.1.2
	            //J1.1.2
	            _.Global.DB_Alarm."word".Line.EmptyLine.Conveyor[_."J1.1.2"].%X1 :=
	            _."ASiGW-MCC001-bw143-C1: Input"."Error J1.1.2";
	            
	        END_REGION
	        
	        // ===== bw143-C1 =====
	        REGION J1.1.3
	            //J1.1.3
	            _.Global.DB_Alarm."word".Line.EmptyLine.Conveyor[_."J1.1.3"].%X1 :=
	            _."ASiGW-MCC001-bw143-C1: Input"."Error J1.1.3";
	            
	        END_REGION
	        
	        // ===== bw143-C1 =====
	        REGION J1.1.4
	            //J1.1.4
	            _.Global.DB_Alarm."word".Line.EmptyLine.Conveyor[_."J1.1.4"].%X1 :=
	            _."ASiGW-MCC001-bw143-C1: Input"."Error J1.1.4";
	            
	        END_REGION
	        
	        // ===== bw143-C1 =====
	        REGION J1.1.5
	            //J1.1.5
	            _.Global.DB_Alarm."word".Line.EmptyLine.Conveyor[_."J1.1.5"].%X1 :=
	            _."ASiGW-MCC001-bw143-C1: Input"."Error J1.1.5";
	            
	        END_REGION
	        
	        // ===== bw143-C1 =====
	        REGION J1.1.6
	            //J1.1.6
	            _.Global.DB_Alarm."word".Line.EmptyLine.Conveyor[_."J1.1.6"].%X1 :=
	            _."ASiGW-MCC001-bw143-C1: Input"."Error J1.1.6";
	            
	        END_REGION
	        
	        // ===== bw143-C1 =====
	        REGION J1.1.7
	            //J1.1.7
	            _.Global.DB_Alarm."word".Line.EmptyLine.Conveyor[_."J1.1.7"].%X1 :=
	            _."ASiGW-MCC001-bw143-C1: Input"."Error J1.1.7";
	            
	        END_REGION
	        
	        // ===== bw143-C1 =====
	        REGION J1.1.8
	            //J1.1.8
	            _.Global.DB_Alarm."word".Line.EmptyLine.Conveyor[_."J1.1.8"].%X1 :=
	            _."ASiGW-MCC001-bw143-C1: Input"."Error J1.1.8";
	            
	        END_REGION
	        
	        // ===== bw143-C1 =====
	        REGION J1.1.9
	            //J1.1.9
	            _.Global.DB_Alarm."word".Line.EmptyLine.Conveyor[_."J1.1.9"].%X1 :=
	            _."ASiGW-MCC001-bw143-C1: Input"."Error J1.1.9";
	            
	        END_REGION
	        
	        // ===== bw143-C1 =====
	        REGION J1.1.10
	            //J1.1.10
	            _.Global.DB_Alarm."word".Line.EmptyLine.Conveyor[_."J1.1.10"].%X1 :=
	            _."ASiGW-MCC001-bw143-C1: Input"."Error J1.1.10";
	            
	        END_REGION
	        
	        // ===== bw143-C1 =====
	        REGION J1.1.11
	            //J1.1.11
	            _.Global.DB_Alarm."word".Line.EmptyLine.Conveyor[_."J1.1.11"].%X1 :=
	            _."ASiGW-MCC001-bw143-C1: Input"."Error J1.1.11";
	            
	        END_REGION
	        
	        // ===== bw143-C1 =====
	        REGION J1.1.12
	            //J1.1.12
	            _.Global.DB_Alarm."word".Line.EmptyLine.Conveyor[_."J1.1.12"].%X1 :=
	            _."ASiGW-MCC001-bw143-C1: Input"."Error J1.1.12";
	            
	        END_REGION
	        
	        // ===== bw143-C1 =====
	        REGION J1.1.13
	            //J1.1.13
	            _.Global.DB_Alarm."word".Line.EmptyLine.Conveyor[_."J1.1.13"].%X1 :=
	            _."ASiGW-MCC001-bw143-C1: Input"."Error J1.1.13";
	            
	        END_REGION
	        
	        // ===== bw143-C1 =====
	        REGION J1.1.14
	            //J1.1.14
	            _.Global.DB_Alarm."word".Line.EmptyLine.Conveyor[_."J1.1.14"].%X1 :=
	            _."ASiGW-MCC001-bw143-C1: Input"."Error J1.1.14";
	            
	        END_REGION
	        
	        // ===== bw143-C1 =====
	        REGION J1.1.15
	            //J1.1.15
	            _.Global.DB_Alarm."word".Line.EmptyLine.Conveyor[_."J1.1.15"].%X1 :=
	            _."ASiGW-MCC001-bw143-C1: Input"."Error J1.1.15";
	            
	        END_REGION
	        
	        // ===== bw143-C1 =====
	        REGION J1.2.1
	            //J1.2.1
	            _.Global.DB_Alarm."word".Line.EmptyLine.Conveyor[_."J1.2.1"].%X1 :=
	            _."ASiGW-MCC001-bw143-C1: Input"."Error J1.2.1";
	            
	        END_REGION
	        
	        // ===== bw143-C1 =====
	        REGION J1.2.2
	            //J1.2.2
	            _.Global.DB_Alarm."word".Line.EmptyLine.Conveyor[_."J1.2.2"].%X1 :=
	            _."ASiGW-MCC001-bw143-C1: Input"."Error J1.2.2";
	            
	        END_REGION
	        
	        // ===== bw143-C1 =====
	        REGION J1.2.3
	            //J1.2.3 Staright for Merger1
	            _.Global.DB_Alarm."word".Line.EmptyLine.Conveyor[_."J1.2.3"].%X1 :=
	            _."ASiGW-MCC001-bw143-C1: Input"."Error J1.2.3";
	            
	        END_REGION
	        
	        // ===== bw143-C1 =====
	        REGION J1.2.4
	            //J1.2.4 Merger 1
	            _.Global.DB_Alarm."word".Line.EmptyLine.Conveyor[_."J1.2.4"].%X1 :=
	            _."ASiGW-MCC001-bw143-C1: Input"."Error J1.2.4";
	            
	        END_REGION
	        
	        // ===== bw143-C1 =====
	        REGION J1.2.5
	            //J1.2.5
	            _.Global.DB_Alarm."word".Line.EmptyLine.Conveyor[_."J1.2.5"].%X1 :=
	            _."ASiGW-MCC001-bw143-C1: Input"."Error J1.2.5";
	            
	        END_REGION
	        
	        // ===== bw143-C1 =====
	        REGION J1.3.1
	            //J1.3.1
	            _.Global.DB_Alarm."word".Line.EmptyLine.Conveyor[_."J1.3.1"].%X1 :=
	            _."ASiGW-MCC001-bw143-C1: Input"."Error J1.3.1";
	            
	        END_REGION
	        
	        // ===== bw143-C1 =====
	        REGION J1.3.2
	            //J1.3.2
	            _.Global.DB_Alarm."word".Line.EmptyLine.Conveyor[_."J1.3.2"].%X1 :=
	            _."ASiGW-MCC001-bw143-C1: Input"."Error J1.3.2";
	            
	        END_REGION
	        
	        // ===== bw143-C1 =====
	        REGION J1.4.1
	            //J1.4.1
	            _.Global.DB_Alarm."word".Line.EmptyLine.Conveyor[_."J1.4.1"].%X1 :=
	            _."ASiGW-MCC001-bw143-C1: Input"."Error J1.4.1";
	            
	        END_REGION
	        
	        // ===== bw143-C1 =====
	        REGION J1.4.2
	            //J1.4.2
	            _.Global.DB_Alarm."word".Line.EmptyLine.Conveyor[_."J1.4.2"].%X1 :=
	            _."ASiGW-MCC001-bw143-C1: Input"."Error J1.4.2";
	            
	        END_REGION
	        
	        // ===== bw143-C1 =====
	        REGION J1.4.3
	            //J1.4.3
	            _.Global.DB_Alarm."word".Line.EmptyLine.Conveyor[_."J1.4.3"].%X1 :=
	            _."ASiGW-MCC001-bw143-C1: Input"."Error J1.4.3";
	            
	        END_REGION
	        
	        // ===== bw143-C1 =====
	        REGION J1.4.4
	            //J1.4.4
	            _.Global.DB_Alarm."word".Line.EmptyLine.Conveyor[_."J1.4.4"].%X1 :=
	            _."ASiGW-MCC001-bw143-C1: Input"."Error J1.4.4";
	            
	        END_REGION
	        
	        // ===== bw143-C1 =====
	        REGION J1.4.5
	            //J1.4.5
	            _.Global.DB_Alarm."word".Line.EmptyLine.Conveyor[_."J1.4.5"].%X1 :=
	            _."ASiGW-MCC001-bw143-C1: Input"."Error J1.4.5";
	            
	        END_REGION
	        
	        // ===== bw143-C1 =====
	        REGION J1.4.6
	            //J1.4.6
	            _.Global.DB_Alarm."word".Line.EmptyLine.Conveyor[_."J1.4.6"].%X1 :=
	            _."ASiGW-MCC001-bw143-C1: Input"."Error J1.4.6";
	            
	        END_REGION
	        
	        // ===== bw143-C1 =====
	        REGION J1.4.7
	            //J1.4.7
	            _.Global.DB_Alarm."word".Line.EmptyLine.Conveyor[_."J1.4.7"].%X1 :=
	            _."ASiGW-MCC001-bw143-C1: Input"."Error J1.4.7";
	            
	        END_REGION
	        
	        // ===== bw143-C1 =====
	        REGION J1.5.1
	            //J1.5.1
	            _.Global.DB_Alarm."word".Line.EmptyLine.Conveyor[_."J1.5.1"].%X1 :=
	            _."ASiGW-MCC001-bw143-C1: Input"."Error J1.5.1";
	            
	        END_REGION
	        
	        // ===== bw143-C1 =====
	        REGION J1.5.2
	            //J1.5.2
	            _.Global.DB_Alarm."word".Line.EmptyLine.Conveyor[_."J1.5.2"].%X1 :=
	            _."ASiGW-MCC001-bw143-C1: Input"."Error J1.5.2";
	            
	        END_REGION
	        
	        // ===== bw143-C1 =====
	        REGION J1.5.3
	            //J1.5.3
	            _.Global.DB_Alarm."word".Line.EmptyLine.Conveyor[_."J1.5.3"].%X1 :=
	            _."ASiGW-MCC001-bw143-C1: Input"."Error J1.5.3";
	            
	        END_REGION
	        
	        // ===== bw143-C1 =====
	        REGION J1.5.4
	            //J1.5.4
	            _.Global.DB_Alarm."word".Line.EmptyLine.Conveyor[_."J1.5.4"].%X1 :=
	            _."ASiGW-MCC001-bw143-C1: Input"."Error J1.5.4";
	            
	        END_REGION
	        
	        // ===== bw143-C1 =====
	        REGION J1.6.1 Mabs
	            //J1.6.1
	            _.Global.DB_Alarm."word".Line.EmptyLine.Conveyor[_."J1.6.1"].%X1 :=
	            _."ASiGW-MCC001-bw143-C1: Input"."J1.6.1 -RemoteOut4";
	            
	        END_REGION
	        
	        // ===== bw143-C1 =====
	        REGION J1.6.1 Mabs
	            //J1.6.1
	            _.Global.DB_Alarm."word".Line.EmptyLine.Conveyor[_."J1.6.2"].%X1 :=
	            _."ASiGW-MCC001-bw143-C1: Input"."J1.6.2 -RemoteOut4";
	            
	        END_REGION
	        
	        
	        // ===== bw143-C1 =====
	        REGION J1.7.1
	            //J1.7.1 (Go straight )
	            _.Global.DB_Alarm."word".Line.EmptyLine.Conveyor[_."J1.7.1"].%X1 :=
	            _."ASiGW-MCC001-bw143-C1: Input"."Error J1.7.1";
	            
	        END_REGION
	        
	        // ===== bw143-C1 =====
	        REGION J1.7.2
	            //J1.7.2
	            _.Global.DB_Alarm."word".Line.EmptyLine.Conveyor[_."J1.7.2"].%X1 :=
	            _."ASiGW-MCC001-bw143-C1: Input"."Error J1.7.2";
	            
	        END_REGION
	        
	        // ===== bw143-C1 =====
	        REGION J1.8.1
	            //J1.8.1
	            _.Global.DB_Alarm."word".Line.EmptyLine.Conveyor[_."J1.8.1"].%X1 :=
	            _."ASiGW-MCC001-bw143-C1: Input"."Error J1.8.1";
	            
	        END_REGION
	        
	        // ===== bw143-C1 =====
	        REGION J1.8.2
	            //J1.8.2
	            _.Global.DB_Alarm."word".Line.EmptyLine.Conveyor[_."J1.8.2"].%X1 :=
	            _."ASiGW-MCC001-bw143-C1: Input"."Error J1.8.2";
	            
	        END_REGION
	        
	        // ===== bw143-C1 =====
	        REGION J1.11.1
	            //J1.11.1
	            _.Global.DB_Alarm."word".Line.EmptyLine.Conveyor[_."J1.11.1"].%X1 :=
	            _."ASiGW-MCC001-bw143-C1: Input"."Error J1.11.1";
	            
	        END_REGION
	        
	        // ===== bw143-C1 =====
	        REGION J1.11.2
	            //J1.11.2
	            _.Global.DB_Alarm."word".Line.EmptyLine.Conveyor[_."J1.11.2"].%X1 :=
	            _."ASiGW-MCC001-bw143-C1: Input"."Error J1.11.2";
	            
	        END_REGION
	        
	        // ===== bw143-C1 =====
	        REGION J1.11.3
	            //J1.11.3
	            _.Global.DB_Alarm."word".Line.EmptyLine.Conveyor[_."J1.11.3"].%X1 :=
	            _."ASiGW-MCC001-bw143-C1: Input"."Error J1.11.3";
	            
	        END_REGION
	        
	        // ===== bw143-C1 =====
	        REGION J1.11.4
	            //J1.11.4
	            _.Global.DB_Alarm."word".Line.EmptyLine.Conveyor[_."J1.11.4"].%X1 :=
	            _."ASiGW-MCC001-bw143-C1: Input"."Error J1.11.4";
	            
	        END_REGION
	        
	        // ===== bw143-C1 =====
	        REGION J1.11.5
	            //J1.11.5
	            _.Global.DB_Alarm."word".Line.EmptyLine.Conveyor[_."J1.11.5"].%X1 :=
	            _."ASiGW-MCC001-bw143-C1: Input"."Error J1.11.5";
	            
	        END_REGION
	        
	        // ===== bw143-C1 =====
	        REGION J1.11.6
	            //J1.11.6
	            _.Global.DB_Alarm."word".Line.EmptyLine.Conveyor[_."J1.11.6"].%X1 :=
	            _."ASiGW-MCC001-bw143-C1: Input"."Error J1.11.6";
	            
	        END_REGION
	        
	        // ===== bw143-C1 =====
	        REGION J1.11.7
	            //J1.11.7
	            _.Global.DB_Alarm."word".Line.EmptyLine.Conveyor[_."J1.11.7"].%X1 :=
	            _."ASiGW-MCC001-bw143-C1: Input"."Error J1.11.7";
	            
	        END_REGION
	        
	        // ===== bw143-C1 =====
	        REGION J1.11.8
	            //J1.11.8
	            _.Global.DB_Alarm."word".Line.EmptyLine.Conveyor[_."J1.11.8"].%X1 :=
	            _."ASiGW-MCC001-bw143-C1: Input"."Error J1.11.8";
	            
	        END_REGION
	        
	        // ===== bw143-C1 =====
	        REGION J1.11.9
	            //J1.11.9
	            _.Global.DB_Alarm."word".Line.EmptyLine.Conveyor[_."J1.11.9"].%X1 :=
	            _."ASiGW-MCC001-bw143-C1: Input"."Error J1.11.9";
	            
	        END_REGION
	        
	        // ===== bw143-C1 =====
	        REGION J1.11.10
	            //J1.11.10
	            _.Global.DB_Alarm."word".Line.EmptyLine.Conveyor[_."J1.11.10"].%X1 :=
	            _."ASiGW-MCC001-bw143-C1: Input"."Error J1.11.10";
	            
	        END_REGION
	        
	        // ===== bw143-C1 =====
	        REGION J1.11.11
	            //J1.11.11
	            _.Global.DB_Alarm."word".Line.EmptyLine.Conveyor[_."J1.11.11"].%X1 :=
	            _."ASiGW-MCC001-bw143-C1: Input"."Error J1.11.11";
	            
	        END_REGION
	        
	        // ===== bw143-C1 =====
	        REGION J1.11.12
	            //J1.11.12
	            _.Global.DB_Alarm."word".Line.EmptyLine.Conveyor[_."J1.11.12"].%X1 :=
	            _."ASiGW-MCC001-bw143-C1: Input"."Error J1.11.12";
	            
	        END_REGION
	        
	        // ===== bw143-C1 =====
	        REGION J1.11.13
	            //J1.11.13
	            _.Global.DB_Alarm."word".Line.EmptyLine.Conveyor[_."J1.11.13"].%X1 :=
	            _."ASiGW-MCC001-bw143-C1: Input"."Error J1.11.13";
	            
	        END_REGION
	        
	        // ===== bw143-C2 =====
	        REGION K1.1.1
	            //K1.1.1
	            _.Global.DB_Alarm."word".Line.EmptyLine.Conveyor[_."K1.1.1"].%X1 :=
	            _."ASiGW-MCC001-bw143-C2: Input"."Error K1.1.1";
	            
	        END_REGION
	        
	        // ===== bw143-C2 =====
	        REGION K1.3.1
	            //K1.3.1
	            _.Global.DB_Alarm."word".Line.EmptyLine.Conveyor[_."K1.3.1"].%X1 :=
	            _."ASiGW-MCC001-bw143-C2: Input"."Error K1.3.1";
	            
	        END_REGION
	        
	        // ===== bw143-C2 =====
	        REGION K1.4.1
	            //K1.4.1
	            _.Global.DB_Alarm."word".Line.EmptyLine.Conveyor[_."K1.4.1"].%X1 :=
	            _."ASiGW-MCC001-bw143-C2: Input"."Error K1.4.1";
	            
	        END_REGION
	        
	        // ===== bw143-C2 =====
	        REGION K1.4.2
	            //K1.4.2
	            _.Global.DB_Alarm."word".Line.EmptyLine.Conveyor[_."K1.4.2"].%X1 :=
	            _."ASiGW-MCC001-bw143-C2: Input"."Error K1.4.2";
	            
	        END_REGION
	        
	        // ===== bw143-C2 =====
	        REGION K1.4.3
	            //K1.4.3
	            _.Global.DB_Alarm."word".Line.EmptyLine.Conveyor[_."K1.4.3"].%X1 :=
	            _."ASiGW-MCC001-bw143-C2: Input"."Error K1.4.3";
	            
	        END_REGION
	        
	        // ===== bw143-C2 =====
	        REGION K1.4.4
	            //K1.4.4
	            _.Global.DB_Alarm."word".Line.EmptyLine.Conveyor[_."K1.4.4"].%X1 :=
	            _."ASiGW-MCC001-bw143-C2: Input"."Error K1.4.4";
	            
	        END_REGION
	        
	        // ===== bw143-C2 =====
	        REGION K1.4.5
	            //K1.4.5
	            _.Global.DB_Alarm."word".Line.EmptyLine.Conveyor[_."K1.4.5"].%X1 :=
	            _."ASiGW-MCC001-bw143-C2: Input"."Error K1.4.5";
	            
	        END_REGION
	        
	        // ===== bw143-C2 =====
	        REGION K1.4.6
	            //K1.4.6
	            _.Global.DB_Alarm."word".Line.EmptyLine.Conveyor[_."K1.4.6"].%X1 :=
	            _."ASiGW-MCC001-bw143-C2: Input"."Error K1.4.6";
	            
	        END_REGION
	        
	        // ===== bw143-C2 =====
	        REGION K1.4.7
	            //K1.4.7
	            _.Global.DB_Alarm."word".Line.EmptyLine.Conveyor[_."K1.4.7"].%X1 :=
	            _."ASiGW-MCC001-bw143-C2: Input"."Error K1.4.7";
	            
	        END_REGION
	        
	        // ===== bw143-C2 =====
	        REGION K1.4.8
	            //K1.4.8
	            _.Global.DB_Alarm."word".Line.EmptyLine.Conveyor[_."K1.4.8"].%X1 :=
	            _."ASiGW-MCC001-bw143-C2: Input"."Error K1.4.8";
	            
	        END_REGION
	        
	        // ===== bw143-C2 =====
	        REGION K1.4.9
	            //K1.4.9
	            _.Global.DB_Alarm."word".Line.EmptyLine.Conveyor[_."K1.4.9"].%X1 :=
	            _."ASiGW-MCC001-bw143-C2: Input"."Error K1.4.9";
	            
	        END_REGION
	        
	        // ===== bw143-C2 =====
	        REGION K1.4.10
	            //K1.4.10
	            _.Global.DB_Alarm."word".Line.EmptyLine.Conveyor[_."K1.4.10"].%X1 :=
	            _."ASiGW-MCC001-bw143-C2: Input"."Error K1.4.10";
	            
	        END_REGION
	        
	        // ===== bw143-C2 =====
	        REGION K1.5.1
	            //K1.5.1
	            _.Global.DB_Alarm."word".Line.EmptyLine.Conveyor[_."K1.5.1"].%X1 :=
	            _."ASiGW-MCC001-bw143-C2: Input"."Error K1.5.1";
	            
	        END_REGION
	        
	        // ===== bw143-C2 =====
	        REGION K1.5.2
	            //K1.5.2
	            _.Global.DB_Alarm."word".Line.EmptyLine.Conveyor[_."K1.5.2"].%X1 :=
	            _."ASiGW-MCC001-bw143-C2: Input"."Error K1.5.2";
	            
	        END_REGION
	        
	        // ===== bw143-C2 =====
	        REGION K1.5.3
	            //K1.5.3
	            _.Global.DB_Alarm."word".Line.EmptyLine.Conveyor[_."K1.5.3"].%X1 :=
	            _."ASiGW-MCC001-bw143-C2: Input"."Error K1.5.3";
	            
	        END_REGION
	        
	        // ===== bw143-C2 =====
	        REGION K1.5.4
	            //K1.5.4
	            _.Global.DB_Alarm."word".Line.EmptyLine.Conveyor[_."K1.5.4"].%X1 :=
	            _."ASiGW-MCC001-bw143-C2: Input"."Error K1.5.4";
	            
	        END_REGION
	        
	        // ===== bw143-C2 =====
	        REGION K1.5.5
	            //K1.5.5
	            _.Global.DB_Alarm."word".Line.EmptyLine.Conveyor[_."K1.5.5"].%X1 :=
	            _."ASiGW-MCC001-bw143-C2: Input"."Error K1.5.5";
	            
	        END_REGION
	        
	        // ===== bw143-C2 =====
	        REGION K1.5.6
	            //K1.5.6
	            _.Global.DB_Alarm."word".Line.EmptyLine.Conveyor[_."K1.5.6"].%X1 :=
	            _."ASiGW-MCC001-bw143-C2: Input"."Error K1.5.6";
	            
	        END_REGION
	        
	        // ===== bw143-C2 =====
	        REGION K1.5.7
	            //K1.5.7
	            _.Global.DB_Alarm."word".Line.EmptyLine.Conveyor[_."K1.5.7"].%X1 :=
	            _."ASiGW-MCC001-bw143-C2: Input"."Error K1.5.7";
	            
	        END_REGION
	        
	        // ===== bw143-C2 =====
	        REGION K1.5.8
	            //K1.5.8
	            _.Global.DB_Alarm."word".Line.EmptyLine.Conveyor[_."K1.5.8"].%X1 :=
	            _."ASiGW-MCC001-bw143-C2: Input"."Error K1.5.8";
	            
	        END_REGION
	        
	        // ===== bw143-C2 =====
	        REGION K1.7.1
	            //K1.7.1
	            _.Global.DB_Alarm."word".Line.EmptyLine.Conveyor[_."K1.7.1"].%X1 :=
	            _."ASiGW-MCC001-bw143-C2: Input"."Error K1.7.1";
	            
	        END_REGION
	        
	        // ===== bw143-C2 =====
	        REGION K1.7.2
	            //K1.7.2
	            _.Global.DB_Alarm."word".Line.EmptyLine.Conveyor[_."K1.7.2"].%X1 :=
	            _."ASiGW-MCC001-bw143-C2: Input"."Error K1.7.2";
	            
	        END_REGION
	        
	        // ===== bw143-C2 =====
	        REGION K1.8.1
	            //K1.8.1
	            _.Global.DB_Alarm."word".Line.EmptyLine.Conveyor[_."K1.8.1"].%X1 :=
	            _."ASiGW-MCC001-bw143-C2: Input"."Error K1.8.1";
	            
	        END_REGION
	        
	        // ===== bw143-C2 =====
	        REGION K1.8.2
	            //K1.8.2
	            _.Global.DB_Alarm."word".Line.EmptyLine.Conveyor[_."K1.8.2"].%X1 :=
	            _."ASiGW-MCC001-bw143-C2: Input"."Error K1.8.2";
	            
	        END_REGION
	        
	        // ===== bw143-C2 =====
	        REGION K1.8.3
	            //K1.8.3
	            _.Global.DB_Alarm."word".Line.EmptyLine.Conveyor[_."K1.8.3"].%X1 :=
	            _."ASiGW-MCC001-bw143-C2: Input"."Error K1.8.3";
	            
	        END_REGION
	        
	        // ===== bw143-C2 =====
	        REGION K1.9.1
	            //K1.9.1
	            _.Global.DB_Alarm."word".Line.EmptyLine.Conveyor[_."K1.9.1"].%X1 :=
	            _."ASiGW-MCC001-bw143-C2: Input"."Error K1.9.1";
	            
	        END_REGION
	        
	        // ===== bw143-C2 =====
	        REGION K1.9.2
	            //K1.9.2
	            _.Global.DB_Alarm."word".Line.EmptyLine.Conveyor[_."K1.9.2"].%X1 :=
	            _."ASiGW-MCC001-bw143-C2: Input"."Error K1.9.2";
	            
	        END_REGION
	        
	        // ===== bw143-C2 =====
	        REGION K1.9.3
	            //K1.9.3
	            _.Global.DB_Alarm."word".Line.EmptyLine.Conveyor[_."K1.9.3"].%X1 :=
	            _."ASiGW-MCC001-bw143-C2: Input"."Error K1.9.3";
	            
	        END_REGION
	        
	        // ===== bw143-C2 =====
	        REGION K1.9.4
	            //K1.9.4
	            _.Global.DB_Alarm."word".Line.EmptyLine.Conveyor[_."K1.9.4"].%X1 :=
	            _."ASiGW-MCC001-bw143-C2: Input"."Error K1.9.4";
	            
	        END_REGION
	        
	        // ===== bw143-C2 =====
	        REGION K1.9.5
	            //K1.9.5
	            _.Global.DB_Alarm."word".Line.EmptyLine.Conveyor[_."K1.9.5"].%X1 :=
	            _."ASiGW-MCC001-bw143-C2: Input"."Error K1.9.5";
	            
	        END_REGION
	        
	        // ===== bw143-C2 =====
	        REGION K1.9.6
	            //K1.9.6
	            _.Global.DB_Alarm."word".Line.EmptyLine.Conveyor[_."K1.9.6"].%X1 :=
	            _."ASiGW-MCC001-bw143-C2: Input"."Error K1.9.6";
	            
	        END_REGION
	        
	        // ===== bw143-C2 =====
	        REGION K1.9.7
	            //K1.9.7
	            _.Global.DB_Alarm."word".Line.EmptyLine.Conveyor[_."K1.9.7"].%X1 :=
	            _."ASiGW-MCC001-bw143-C2: Input"."Error K1.9.7";
	            
	        END_REGION
	        
	        // ===== bw143-C2 =====
	        REGION K1.10.1
	            //K1.10.1
	            _.Global.DB_Alarm."word".Line.EmptyLine.Conveyor[_."K1.10.1"].%X1 :=
	            _."ASiGW-MCC001-bw143-C2: Input"."Error K1.10.1";
	            
	        END_REGION
	        
	        // ===== bw200-C2 =====
	        REGION J2.1.1
	            //J2.1.1
	            _.Global.DB_Alarm."word".Line.EmptyLine.Conveyor[_."J2.1.1"].%X1 :=
	            _."ASiGW-MCC001-bw200-C2: Input"."Error J2.1.1";
	            
	        END_REGION
	        
	        // ===== bw200-C2 =====
	        REGION J2.1.2
	            //J2.1.2
	            _.Global.DB_Alarm."word".Line.EmptyLine.Conveyor[_."J2.1.2"].%X1 :=
	            _."ASiGW-MCC001-bw200-C2: Input"."Error J2.1.2";
	            
	        END_REGION
	        
	        // ===== bw200-C2 =====
	        REGION J2.1.3
	            //J2.1.3
	            _.Global.DB_Alarm."word".Line.EmptyLine.Conveyor[_."J2.1.3"].%X1 :=
	            _."ASiGW-MCC001-bw200-C2: Input"."Error J2.1.3";
	            
	        END_REGION
	        
	        // ===== bw200-C2 =====
	        REGION J2.1.4
	            //J2.1.4
	            _.Global.DB_Alarm."word".Line.EmptyLine.Conveyor[_."J2.1.4"].%X1 :=
	            _."ASiGW-MCC001-bw200-C2: Input"."Error J2.1.4";
	            
	        END_REGION
	        
	        // ===== bw200-C2 =====
	        REGION J2.1.5
	            //J2.1.5
	            _.Global.DB_Alarm."word".Line.EmptyLine.Conveyor[_."J2.1.5"].%X1 :=
	            _."ASiGW-MCC001-bw200-C2: Input"."Error J2.1.5";
	            
	        END_REGION
	        
	        // ===== bw200-C2 =====
	        REGION J2.1.6
	            //J2.1.6
	            _.Global.DB_Alarm."word".Line.EmptyLine.Conveyor[_."J2.1.6"].%X1 :=
	            _."ASiGW-MCC001-bw200-C2: Input"."Error J2.1.6";
	            
	        END_REGION
	        
	        // ===== bw200-C2 =====
	        REGION J2.1.7
	            //J2.1.7
	            _.Global.DB_Alarm."word".Line.EmptyLine.Conveyor[_."J2.1.7"].%X1 :=
	            _."ASiGW-MCC001-bw200-C2: Input"."Error J2.1.7";
	            
	        END_REGION
	        
	        // ===== bw200-C2 =====
	        REGION J2.1.8
	            //J2.1.8
	            _.Global.DB_Alarm."word".Line.EmptyLine.Conveyor[_."J2.1.8"].%X1 :=
	            _."ASiGW-MCC001-bw200-C2: Input"."Error J2.1.8";
	            
	        END_REGION
	        
	        // ===== bw200-C2 =====
	        REGION J2.1.9
	            //J2.1.9
	            _.Global.DB_Alarm."word".Line.EmptyLine.Conveyor[_."J2.1.9"].%X1 :=
	            _."ASiGW-MCC001-bw200-C2: Input"."Error J2.1.9";
	            
	        END_REGION
	        
	        // ===== bw200-C2 =====
	        REGION J2.1.10
	            //J2.1.10
	            _.Global.DB_Alarm."word".Line.EmptyLine.Conveyor[_."J2.1.10"].%X1 :=
	            _."ASiGW-MCC001-bw200-C2: Input"."Error J2.1.10";
	            
	        END_REGION
	        
	        // ===== bw200-C2 =====
	        REGION J2.1.11
	            //J2.1.11
	            _.Global.DB_Alarm."word".Line.EmptyLine.Conveyor[_."J2.1.11"].%X1 :=
	            _."ASiGW-MCC001-bw200-C2: Input"."Error J2.1.11";
	            
	        END_REGION
	        
	        // ===== bw200-C2 =====
	        REGION J2.1.12
	            //J2.1.12
	            _.Global.DB_Alarm."word".Line.EmptyLine.Conveyor[_."J2.1.12"].%X1 :=
	            _."ASiGW-MCC001-bw200-C2: Input"."Error J2.1.12";
	            
	        END_REGION
	        
	        // ===== bw200-C2 =====
	        REGION J2.1.13
	            //J2.1.13
	            _.Global.DB_Alarm."word".Line.EmptyLine.Conveyor[_."J2.1.13"].%X1 :=
	            _."ASiGW-MCC001-bw200-C2: Input"."Error J2.1.13";
	            
	        END_REGION
	        
	        // ===== bw200-C2 =====
	        REGION J2.1.14
	            //J2.1.14
	            _.Global.DB_Alarm."word".Line.EmptyLine.Conveyor[_."J2.1.14"].%X1 :=
	            _."ASiGW-MCC001-bw200-C2: Input"."Error J2.1.14";
	            
	        END_REGION
	        
	        // ===== bw200-C2 =====
	        REGION J2.1.15
	            //J2.1.15
	            _.Global.DB_Alarm."word".Line.EmptyLine.Conveyor[_."J2.1.15"].%X1 :=
	            _."ASiGW-MCC001-bw200-C2: Input"."Error J2.1.15";
	            
	        END_REGION
	        
	        // ===== bw200-C2 =====
	        REGION J2.2.1
	            //J2.2.1
	            _.Global.DB_Alarm."word".Line.EmptyLine.Conveyor[_."J2.2.1"].%X1 :=
	            _."ASiGW-MCC001-bw200-C2: Input"."Error J2.2.1";
	            
	        END_REGION
	        
	        // ===== bw200-C2 =====
	        REGION J2.2.2
	            //J2.2.2
	            _.Global.DB_Alarm."word".Line.EmptyLine.Conveyor[_."J2.2.2"].%X1 :=
	            _."ASiGW-MCC001-bw200-C2: Input"."Error J2.2.2";
	            
	        END_REGION
	        
	        // ===== bw200-C2 =====
	        REGION J2.4.1
	            //J2.4.1 Arm for Merger1
	            _.Global.DB_Alarm."word".Line.EmptyLine.Conveyor[_."J2.4.1"].%X1 :=
	            _."ASiGW-MCC001-bw200-C2: Input"."Error J2.4.1";
	            
	        END_REGION
	        
	        
	    END_IF;
	END_REGION
	
	
	
	
	
	
	
	
	
	
END_FUNCTION
END_NAMESPACE

NAMESPACE EmptyLine
FUNCTION FC_SimuAlarm : Void
{ S7_Optimized_Access := 'TRUE' ; Published := 'FALSE' }
VERSION : 0.1
   VAR_TEMP 
      cmp : Struct
         Line : Struct
            B1 : Array[_.minEmptyLine.._.maxEmptyLine] of Bool;
         END_STRUCT;
      END_STRUCT;
   END_VAR


BEGIN
	// ==========================================================================================================================================
	// Company        : LogTech, s.r.o.
	// Created by     : Anton Vinoth Soundraraj
	// Block          : FC_SimuAlarm
	// Project        : Lékarna DC Chrudim
	// Project number : 23-157
	// ==========================================================================================================================================
	
	
	REGION Simulation active alarm
	    
	    (* REGION Line B1
	        
	    // if any of the simulation trigger fault is active
	        _.LineB1.DB_Alarm.Simu.%X0 := NOT (#cmp.Line.B1 ="DB_SystemSimu".TriggerFault.Line.ProductionTote.Conveyor);
	    // if any of the simulation trigger sensor is active
	        _.LineB1.DB_Alarm.Simu.%X1 := NOT (#cmp.Line.B1 ="DB_SystemSimu".TriggerSensor.Line.ProductionTote.Conveyor);
	        
	    END_REGION *)
	    
	END_REGION
	
	REGION Fire bit
	    
	    (* // if simulation fire signal is active
	    "DB_Alarm".Simu.%X6 := "DB_SystemSimu".Fire; *)
	    
	END_REGION
	
	
	
	
	
	
	
END_FUNCTION
END_NAMESPACE

NAMESPACE Global
FUNCTION FC_ReadSystemSSR : Void
{ S7_Optimized_Access := 'TRUE' ; Published := 'FALSE' }
VERSION : 0.1

BEGIN
	// ==========================================================================================================================================
	// Company        : LogTech, s.r.o.
	// Created by     : Anton Vinoth Soundraraj
	// Block          : FC_ReadSystemSSR
	// Project        : Lékarna DC Chrudim
	// Project number : 23-157
	// ==========================================================================================================================================
	
	REGION ProductionLine
	    
	    // Start Stop Reset IO
	    
	    // Activate Start bit
	    //DB_SystemSSR.Line.ProductionLine.StartSystem :=
	    DB_SystemSSR.Zone."1".StartSystem :=
	    DB_SystemSSR.FromHMI.Line.ProductionLine.StartSystem OR 
	    _.DB_Sync.startbit1;
	    // Activate Stop bit
	    DB_SystemSSR.Zone."1".StopSystem :=
	    DB_SystemSSR.FromHMI.Line.ProductionLine.StopSystem OR
	    _.DB_Sync.stopbit1;
	    // Activate Reset bit
	    DB_SystemSSR.Zone."1".ResetSystem :=
	    DB_SystemSSR.FromHMI.Line.ProductionLine.ResetSystem OR
	    _.DB_Sync.resetbit1;
	    
	END_REGION
	
	REGION EmptyLine
	    
	    // Start Stop Reset IO
	    
	    // Activate Start bit
	    DB_SystemSSR.Zone."2".StartSystem :=
	    DB_SystemSSR.FromHMI.Line.EmptyLine.StartSystem OR
	    _.DB_Sync.startbit2;
	    // Activate Stop bit
	    DB_SystemSSR.Zone."2".StopSystem :=
	    DB_SystemSSR.FromHMI.Line.EmptyLine.StopSystem OR
	    _.DB_Sync.stopbit2;
	    // Activate Reset bit
	    DB_SystemSSR.Zone."2".ResetSystem :=
	    DB_SystemSSR.FromHMI.Line.EmptyLine.ResetSystem OR
	    _.DB_Sync.resetbit2;
	    
	END_REGION
	(*
	REGION PackedLine
	    
	    // Start Stop Reset IO
	    
	    // Activate Start bit
	    DB_SystemSSR.Line.PackedLine.StartSystem :=
	    DB_SystemSSR.FromHMI.Line.PackedLine.StartSystem OR
	    _.DB_Sync.startbit;
	    // Activate Stop bit
	    DB_SystemSSR.Line.PackedLine.StopSystem :=
	    DB_SystemSSR.FromHMI.Line.PackedLine.StopSystem OR
	    _.DB_Sync.stopbit;
	    // Activate Reset bit
	    DB_SystemSSR.Line.PackedLine.ResetSystem :=
	    DB_SystemSSR.FromHMI.Line.PackedLine.ResetSystem OR
	    _.DB_Sync.resetbit;
	    
	END_REGION
 automatically inserted *)
END_FUNCTION
END_NAMESPACE

NAMESPACE Global
FUNCTION_BLOCK FB_Conveyor
{ S7_Optimized_Access := 'TRUE' ; Published := 'TRUE' }
VERSION : 0.1
   VAR_INPUT 
      ConveyorID : Int;
      ConveyorSensor : Bool;
      Fault : Bool;
      Upstream : Bool;
      Downstream : Bool;
      Interlock : Bool;
   END_VAR

   VAR_OUTPUT 
      RunForward : Bool;
      WriteAsiDir : Bool;
      WriteAsiSpeed : Bool;
      NordControlEnable : Word;
      NordSetpoint : Word;
      ImcSpeed : SInt;
   END_VAR

   VAR 
      sConvID : Int;
      ReadInputSignal : Struct
         ConveyorSensor : Bool;
         EmergencyStop : Bool;
         Fault : Bool;
      END_STRUCT;
      MotorType : Struct
         "24v-ASi" : Bool;
         nord : Bool;
         "24v-IMC" : Bool;
      END_STRUCT;
      Active : Struct
         Line : Struct
            ProductionLine : Bool;
            EmptyLine : Bool;
            PackedLine : Bool;
         END_STRUCT;
         EstopZone { S7_SetPoint := 'False'} : EsopZone;
      END_STRUCT;
      CONVEYOR_SENSOR : FB_Sensor;
      CONVEYOR_SENSOR_BLOCKAGE : FB_SensorBlockage;
      CONVEYOR_STATUS_ON : FB_StatusON;
      CONVEYOR_STATUS_READY : FB_StatusReady;
      CONVEYOR_STATUS_FAULT : FB_StatusFault;
      "RUN/STOP_CONVEYOR" : FB_RunStop;
      ENERGY_SAVE : FB_EnergySave;
      AUTO_RESET : FB_AutoReset;
      SSR { S7_SetPoint := 'False'} : SystemSSR;
      ReadConveyorStatus : ConveyorStatus;
      ReadConveyorParameters { S7_SetPoint := 'False'} : ConveyorParameters := ((), [2(T#10ms)], (), (), (), ());
      ConveyorFault : Fault;
      SimuMode : Struct
         Sensor : Bool;
         Fault : Bool;
         Estop : Struct
            Zone : Struct
               "1" : Bool;
               "2" : Bool;
               "3" : Bool;
               "4" : Bool;
            END_STRUCT;
         END_STRUCT;
      END_STRUCT;
      StartUpTimer {InstructionName := 'TOF_TIME'; LibVersion := '1.0'; S7_SetPoint := 'False'} : TOF_TIME;
      FT_StartUp {InstructionName := 'F_TRIG'; LibVersion := '1.0'} : F_TRIG;
      SetStartUp { S7_SetPoint := 'True'} : Bool;
      FilteredSensor { S7_SetPoint := 'True'} : Bool;
      StopSystemFireActive : Bool;
      EnergySave : Bool;
      StartMotorForward : Bool;
      StartMotorReverse : Bool;
      AutoReset { S7_SetPoint := 'True'} : Bool;
      NullSpeed : SInt;
      VisuColor : Word;
      NordSetpointRun : Word := 16#047F;
      NordSetpointReady : Word := 16#047E;
      NordFaultAck : Word := 16#0080;
   END_VAR


BEGIN
	// ==========================================================================================================================================
	// Company        : LogTech, s.r.o.
	// Created by     : Anton Vinoth Soundraraj
	// Block          : FB_Conveyor
	// Project        : Lékarna DC Chrudim
	// Project number : 23-157
	// ==========================================================================================================================================
	
	// input to static
	#sConvID := #ConveyorID;
	
	REGION Active Line
	    
	    // Production Line
	    IF (#ConveyorID >= _.gminProductionLine AND
	        #ConveyorID <= _.gmaxProductionLine)
	    THEN
	        #Active.Line.ProductionLine := TRUE;
	    END_IF;
	    
	    // Empty Line
	    IF (#ConveyorID >= _.gminEmptyLine AND
	        #ConveyorID <= _.gmaxEmptyLine)
	    THEN
	        #Active.Line.EmptyLine := TRUE;
	    END_IF;
	    
	    // Packed Line
	    IF (#ConveyorID >= _.gminPackedLine AND
	        #ConveyorID <= _.gmaxPackedLine)
	    THEN
	        #Active.Line.PackedLine := TRUE;
	    END_IF;
	    
	END_REGION
	
	REGION Init motor type
	    
	    REGION ASi Motor Type
	        // line Production, Empty and Packed
	        //Production Line
	        IF (#ConveyorID >= _.gminProductionLine AND
	            #ConveyorID <= _.gmaxProductionLine) OR
	            //Empty Line
	            (#ConveyorID >= _.gminEmptyLine AND
	            #ConveyorID <= _.gmaxEmptyLine) OR
	            //Packed line 
	            (#ConveyorID >= _.gminPackedLine AND
	            #ConveyorID <= _.gmaxPackedLine)
	        THEN
	            #MotorType."24v-ASi" := TRUE;
	        END_IF;
	    END_REGION
	
	    REGION InterRoll Motor Type
	        //Packed line 
	        IF (#ConveyorID >= _.gminPackedLine AND
	            #ConveyorID <= _.gmaxPackedLine)
	        THEN
	            #MotorType."24v-IMC" := TRUE;
	        END_IF;
	    END_REGION
	
	    
	END_REGION
	
	REGION Estop zone
	    
	        // Production Line A1
	    IF (#ConveyorID >= _."gA1.1.1" AND
	        #ConveyorID <= _."gA1.7.6") OR
	        (#ConveyorID >= _."gB1.1.1" AND
	        #ConveyorID <= _."gC1.4.2") OR
	       // (#ConveyorID >= _."gA1.6.1" AND
	       // #ConveyorID <= _."gA1.6.2") OR
	       // (#ConveyorID >= _."gB1.6.1" AND
	       // #ConveyorID <= _."gC1.3.1") OR
	        // Empty Line A1
	        (#ConveyorID >= _."gJ1.5.2" AND
	        #ConveyorID <= _."gJ1.6.2")
	    THEN
	        #Active.EstopZone."1" := TRUE;
	    END_IF;
	    
	    // Production Line A2
	    IF  (#ConveyorID >= _."gA1.8.1" AND
	        #ConveyorID <= _."gA2.4.26") OR
	        (#ConveyorID >= _."gD1.1.1" AND
	        #ConveyorID <= _."gE1.6.1") OR
	        //(#ConveyorID >= _."gA1.9.1" AND
	        //#ConveyorID <= _."gA1.9.2") OR
	        //(#ConveyorID >= _."gA1.13.1" AND
	        //#ConveyorID <= _."gA2.1.1") OR
	        //(#ConveyorID >= _."gD1.9.1" AND
	        //#ConveyorID <= _."gD1.10.1") OR
	        //Empty Line A2
	        (#ConveyorID >= _."gJ1.1.1" AND
	        #ConveyorID <= _."gJ1.5.1") OR 
	        // Packed Line
	        (#ConveyorID >= _.gminPackedLine AND
	        #ConveyorID <= _.gmaxPackedLine)
	    THEN
	        #Active.EstopZone."2" := TRUE;
	    END_IF;
	    
	END_REGION
	
	REGION SystemSSR
	    
	    //Zone 1
	    IF #Active.EstopZone."1" THEN
	        #SSR.StartSystem := DB_SystemSSR.Zone."1".StartSystem;
	        #SSR.StopSystem := DB_SystemSSR.Zone."1".StopSystem;
	        #SSR.ResetSystem := DB_SystemSSR.Zone."1".ResetSystem;
	    END_IF;
	    
	    //Zone 2
	    IF #Active.EstopZone."2" THEN
	        #SSR.StartSystem := DB_SystemSSR.Zone."2".StartSystem;
	        #SSR.StopSystem := DB_SystemSSR.Zone."2".StopSystem;
	        #SSR.ResetSystem := DB_SystemSSR.Zone."2".ResetSystem;
	    END_IF;
	    
	END_REGION
	
	REGION Read Simu inputs  
	    
	    // ProductionLine
	    IF #Active.Line.ProductionLine THEN
	        // read simu
	        #SimuMode.Sensor := DB_SystemSimu.TriggerSensor.Line.ProductionLine.Conveyor[#ConveyorID];
	        #SimuMode.Fault := DB_SystemSimu.TriggerFault.Line.ProductionLine.Conveyor[#ConveyorID];
	    END_IF;
	    
	    // EmptyLine
	    IF #Active.Line.EmptyLine THEN
	        // read simu
	        #SimuMode.Sensor := DB_SystemSimu.TriggerSensor.Line.EmptyLine.Conveyor[#ConveyorID];
	        #SimuMode.Fault := DB_SystemSimu.TriggerFault.Line.EmptyLine.Conveyor[#ConveyorID];
	    END_IF;
	    
	    // PackedLine
	    IF #Active.Line.PackedLine THEN
	        // read simu
	        #SimuMode.Sensor := DB_SystemSimu.TriggerSensor.Line.PackedLine.Conveyor[#ConveyorID];
	        #SimuMode.Fault := DB_SystemSimu.TriggerFault.Line.PackedLine.Conveyor[#ConveyorID];
	    END_IF;
	    
	END_REGION
	
	REGION Read Input
	    
	    // read all inputs to the block
	    // Conveyor input read signals
	    #ReadInputSignal.ConveyorSensor := #ConveyorSensor OR   // NOT #ConveyorSensor
	    #SimuMode.Sensor; // simu call
	    #ReadInputSignal.Fault := #Fault OR
	    #SimuMode.Fault; // simu call;
	    #ReadInputSignal.EmergencyStop := // all estop zones are connected together
	    _.DB_SafetyStandard.ToStandard.EstopActive;
	    
	END_REGION
	
	REGION READ AND INIT
	    
	    REGION Init conveyor parameters
	        
	        // Conveyor Parameter
	        // ProductionLine
	        IF #Active.Line.ProductionLine THEN
	            #ReadConveyorParameters := DB_ConveyorParameters.Line.ProductionLine.Conveyor[#ConveyorID];
	        END_IF;
	        // EmptyLine
	        IF #Active.Line.EmptyLine THEN
	            #ReadConveyorParameters := DB_ConveyorParameters.Line.EmptyLine.Conveyor[#ConveyorID];
	        END_IF;
	        // PackedLine
	        IF #Active.Line.PackedLine THEN
	            #ReadConveyorParameters := DB_ConveyorParameters.Line.PackedLine.Conveyor[#ConveyorID];
	        END_IF;
	        
	    END_REGION
	    
	    REGION Sensor Filter
	        
	        // FB_Sensor
	        // called as MIDB
	        
	        #CONVEYOR_SENSOR(Sensor           := #ReadInputSignal.ConveyorSensor,
	                         SensorFilterTime := #ReadConveyorParameters.SensorFilterTime,
	                         FilteredSensor   => #FilteredSensor);
	        
	    END_REGION
	    
	    REGION FIRE
	        
	        // Fire signal from fire system stops the whole system
	        // System can be reset from Fire status only if the fire signal is deactivated
	        
	        // FIRE ALARM ACTIVE --> STOP SYSTEM
	        IF DB_SystemSimu.Fire THEN
	            #StopSystemFireActive := TRUE;
	        END_IF;
	        // RESET --> FIRE ALARM
	        IF #SSR.ResetSystem AND NOT DB_SystemSimu.Fire THEN
	            #StopSystemFireActive := FALSE;
	        END_IF;
	        
	    END_REGION
	    
	END_REGION
	
	REGION Conveyor startup
	    
	    // Conveyor StartUp: Conveyor startup signal after preset time
	    #StartUpTimer.TOF(IN := #SSR.StartSystem,
	                      PT := #ReadConveyorParameters.StartUpTime);
	    
	    #FT_StartUp(CLK := #StartUpTimer.Q);
	    
	    // set startup after the preset
	    #SetStartUp := #FT_StartUp.Q;
	    
	END_REGION
	
	REGION Conveyor Status
	    
	    REGION Status ON
	        
	        // ----------------------------------------->>>>>>> STATUS ON <<<<<<<-----------------------------------------
	        // FB_ConveyorStatusON
	        // called as IDMB
	        
	        #CONVEYOR_STATUS_ON(SystemStartActive := #SSR.StartSystem,
	                            StatusStop        := #ReadConveyorStatus.Stop,
	                            StatusEStop       := #ReadConveyorStatus.Estop,
	                            StatusManual      := #ReadConveyorStatus.Manual,
	                            StatusFault       := #ReadConveyorStatus.Fault,
	                            FireAlarmActive   := #StopSystemFireActive,
	                            StatusON          => #ReadConveyorStatus.ON);
	        
	    END_REGION
	    
	    REGION Status Ready
	        
	        // ----------------------------------------->>>>>>> STATUS READY <<<<<<<-----------------------------------------
	        // FB_ConveyorStatusReady
	        // called as MIDB
	        
	        #CONVEYOR_STATUS_READY(StatusON        := #ReadConveyorStatus.ON,
	                               StatusESTOP     := #ReadConveyorStatus.Estop,
	                               StatusFAULT     := #ReadConveyorStatus.Fault,
	                               StatusMAN       := #ReadConveyorStatus.Manual,
	                               SignalFIRE      := #StopSystemFireActive,
	                               SystemAlertTime := #ReadConveyorParameters.StartUpTime,
	                               StatusReady     => #ReadConveyorStatus.ReadytoRun);
	        
	    END_REGION
	    
	    REGION Status Occupied
	        
	        // ----------------------------------------->>>>>>> STATUS OCCUPIED <<<<<<<-----------------------------------------
	        #ReadConveyorStatus.Occupied := #FilteredSensor;
	        
	    END_REGION
	    
	    REGION Status Running
	        
	        // ----------------------------------------->>>>>>> STATUS RUNNING <<<<<<<-----------------------------------------
	        
	        #ReadConveyorStatus.Running := #StartMotorForward OR #StartMotorReverse;
	        
	    END_REGION
	    
	    REGION Status Fault
	        
	        // ----------------------------------------->>>>>>> STATUS FAULT <<<<<<<-----------------------------------------
	        
	        // Automatic reset trigger to the needed drive after wakeup from ESTOP power miss (only if needed)
	        // will trigger for every Reset active
	        
	        #AUTO_RESET(AckIN := #SSR.ResetSystem,
	                    Ack   => #AutoReset);
	        
	        // Reading error signal from the motor drive
	        #ConveyorFault.Motor_Error := #ReadInputSignal.Fault;
	        
	        // FC_ConveyorStatusFault
	        #CONVEYOR_STATUS_FAULT(FaultActive   := #ConveyorFault.Motor_Error,
	                               ResetFault    := #SSR.ResetSystem OR #AutoReset,
	                               StatusRunning := #ReadConveyorStatus.Running,
	                               FaultStatus   => #ReadConveyorStatus.Fault);
	        
	    END_REGION
	    
	    REGION Status ESTOP
	        
	        // ----------------------------------------->>>>>>> STATUS ESTOP <<<<<<<-----------------------------------------
	        
	        // EMERGENCY STOP ACTIVE --> STOP SYSTEM
	        IF #ReadInputSignal.EmergencyStop THEN
	            #ReadConveyorStatus.Estop := TRUE;
	        END_IF;
	        // RESET --> EMERGENCY STOP
	        IF #AutoReset AND NOT #ReadInputSignal.EmergencyStop THEN // (reset after 12 seconds) : Auto Reset
	            #ReadConveyorStatus.Estop := FALSE;
	        END_IF;
	        
	    END_REGION
	    
	    REGION Status Manual
	        
